	(*Part 17 Present*)
		Part_Present17FB(
			Sensor_Input:= N03.I.0,
			On_Trigger1:= Enable_Motion AND In_Auto AND NOT Unload_Complete AND (Model_ID <> 1) AND Repo_Reqs.0,
			On_Trigger2:= TRUE,
			Off_Trigger1:= Dry_Cycle OR (Cycle_Complete  AND NOT Enable_Motion),
			Off_Trigger2:= TRUE,
			Disable_Faults:= Dry_Cycle OR (Weld_Robots_WorkingOK) OR Turntable_Bypassed,
			Fault_Delay:= T#1.5s,
			Status=> Part_Present17,
			Faulted=>  PPFaults.17);

	(*Part 18 Present*)
		Part_Present18FB(
			Sensor_Input:= N03.I.1,
			On_Trigger1:= Enable_Motion AND In_Auto AND NOT Unload_Complete AND (Model_ID>3),
			On_Trigger2:= TRUE,
			Off_Trigger1:= Dry_Cycle OR (Cycle_Complete  AND NOT Enable_Motion),
			Off_Trigger2:= TRUE,
			Disable_Faults:= Dry_Cycle OR (Weld_Robots_WorkingOK) OR Turntable_Bypassed,
			Fault_Delay:= T#1.5s,
			Status=> Part_Present18,
			Faulted=>  PPFaults.18);

	(*Part 19 Present*)
		Part_Present19FB(
			Sensor_Input:= N03.I.2,
			On_Trigger1:= Enable_Motion AND In_Auto AND NOT Unload_Complete AND NOT Welding_Complete,
			On_Trigger2:= TRUE,
			Off_Trigger1:= Dry_Cycle OR (Cycle_Complete  AND NOT Enable_Motion),
			Off_Trigger2:= TRUE,
			Disable_Faults:= Dry_Cycle OR (Weld_Robots_WorkingOK) OR Turntable_Bypassed,
			Fault_Delay:= T#1.5s,
			Status=> Part_Present19,
			Faulted=>  PPFaults.19);

	(*Part 20 Present*)
		Part_Present20FB(
			Sensor_Input:= N03.I.3,
			On_Trigger1:= Enable_Motion AND In_Auto AND NOT Unload_Complete,
			On_Trigger2:= TRUE,
			Off_Trigger1:= Dry_Cycle OR (Cycle_Complete  AND NOT Enable_Motion),
			Off_Trigger2:= TRUE,
			Disable_Faults:= Dry_Cycle OR (Weld_Robots_WorkingOK) OR Turntable_Bypassed,
			Fault_Delay:= T#1.5s,
			Status=> Part_Present20,
			Faulted=>  PPFaults.20);

	(*Part 21 Present*)
		Part_Present21FB(
			Sensor_Input:= N03.I.4,
			On_Trigger1:= Enable_Motion AND In_Auto AND NOT Unload_Complete AND NOT Welding_Complete,
			On_Trigger2:= TRUE,
			Off_Trigger1:= Dry_Cycle OR (Cycle_Complete  AND NOT Enable_Motion),
			Off_Trigger2:= TRUE,
			Disable_Faults:= Dry_Cycle OR (Weld_Robots_WorkingOK) OR Turntable_Bypassed,
			Fault_Delay:= T#1.5s,
			Status=> Part_Present21,
			Faulted=>  PPFaults.21);

	(*Part 22 Present*)
		Part_Present22FB(
			Sensor_Input:= N03.I.5,
			On_Trigger1:= Enable_Motion AND In_Auto AND NOT Unload_Complete AND (Model_ID=3) AND NOT Welding_Complete,
			On_Trigger2:= TRUE,
			Off_Trigger1:= Dry_Cycle OR (Cycle_Complete  AND NOT Enable_Motion),
			Off_Trigger2:= TRUE,
			Disable_Faults:= Dry_Cycle OR (Weld_Robots_WorkingOK) OR Turntable_Bypassed,
			Fault_Delay:= T#1.5s,
			Status=> Part_Present22,
			Faulted=>  PPFaults.22);

	(*Part 23 Present - should always be off, detects wrong part loaded*)
		Part_Present23FB(
			Sensor_Input:= N03.I.6,
			On_Trigger1:= FALSE,
			On_Trigger2:= TRUE,
			Off_Trigger1:= Enable_Motion AND In_Auto AND NOT Unload_Complete,
			Off_Trigger2:= TRUE,
			Disable_Faults:= Dry_Cycle OR (Weld_Robots_WorkingOK) OR Turntable_Bypassed,
			Fault_Delay:= T#1.5s,
			Status=> Part_Present23,
			Faulted=>  PPFaults.23);

	(*Part 24 Present*)
		Part_Present24FB(
			Sensor_Input:= N03.I.7,
			On_Trigger1:= Enable_Motion AND In_Auto AND NOT Unload_Complete AND (Model_ID = 2),
			On_Trigger2:= TRUE,
			Off_Trigger1:= Dry_Cycle OR (Cycle_Complete  AND NOT Enable_Motion),
			Off_Trigger2:= TRUE,
			Disable_Faults:= Dry_Cycle OR (Weld_Robots_WorkingOK) OR Turntable_Bypassed,
			Fault_Delay:= T#1.5s,
			Status=> Part_Present24,
			Faulted=>  PPFaults.24);

	(*Part 25 Present*)
		Part_Present25FB(
			Sensor_Input:= N04.I.0,
			On_Trigger1:= Enable_Motion AND In_Auto AND NOT Unload_Complete,
			On_Trigger2:= TRUE,
			Off_Trigger1:= Dry_Cycle OR (Cycle_Complete  AND NOT Enable_Motion),
			Off_Trigger2:= TRUE,
			Disable_Faults:= Dry_Cycle OR (Weld_Robots_WorkingOK) OR Turntable_Bypassed,
			Fault_Delay:= T#1.5s,
			Status=> Part_Present25,
			Faulted=>  PPFaults.25);

	(*Part 26 Present*)
		Part_Present26FB(
			Sensor_Input:= N04.I.1,
			On_Trigger1:= Enable_Motion AND In_Auto AND NOT Unload_Complete,
			On_Trigger2:= TRUE,
			Off_Trigger1:= Dry_Cycle OR (Cycle_Complete  AND NOT Enable_Motion),
			Off_Trigger2:= TRUE,
			Disable_Faults:= Dry_Cycle OR (Weld_Robots_WorkingOK) OR Turntable_Bypassed,
			Fault_Delay:= T#1.5s,
			Status=> Part_Present26,
			Faulted=>  PPFaults.26);

	(*Part 27 Present*)
		Part_Present27FB(
			Sensor_Input:= N04.I.2,
			On_Trigger1:= Enable_Motion AND In_Auto AND NOT Unload_Complete AND NOT Welding_Complete,
			On_Trigger2:= TRUE,
			Off_Trigger1:= Dry_Cycle OR (Cycle_Complete  AND NOT Enable_Motion),
			Off_Trigger2:= TRUE,
			Disable_Faults:= Dry_Cycle OR (Weld_Robots_WorkingOK) OR Turntable_Bypassed,
			Status=> Part_Present27,
			Faulted=>  PPFaults.27);
			
	(*Part 28 Present*)
		Part_Present28FB(
			Sensor_Input:= N04.I.3,
			On_Trigger1:= Enable_Motion AND In_Auto AND NOT Unload_Complete,
			On_Trigger2:= TRUE,
			Off_Trigger1:= Dry_Cycle OR (Cycle_Complete  AND NOT Enable_Motion),
			Off_Trigger2:= TRUE,
			Disable_Faults:= Dry_Cycle OR (Weld_Robots_WorkingOK) OR Turntable_Bypassed,
			Fault_Delay:= T#1.5s,
			Status=> Part_Present28,
			Faulted=>  PPFaults.28);

	(*Part 29 Present*)
		Part_Present29FB(
			Sensor_Input:= N04.I.4,
			On_Trigger1:= Enable_Motion AND In_Auto AND NOT Unload_Complete,
			On_Trigger2:= TRUE,
			Off_Trigger1:= Dry_Cycle OR (Cycle_Complete  AND NOT Enable_Motion),
			Off_Trigger2:= TRUE,
			Disable_Faults:= Dry_Cycle OR (Weld_Robots_WorkingOK) OR Turntable_Bypassed,
			Fault_Delay:= T#1.5s,
			Status=> Part_Present29,
			Faulted=>  PPFaults.29);

	(*Part 30 Present*)
		Part_Present30FB(
			Sensor_Input:= N04.I.5,
			On_Trigger1:= Enable_Motion AND In_Auto AND NOT Unload_Complete AND (Model_ID=7),
			On_Trigger2:= TRUE,
			Off_Trigger1:= Dry_Cycle OR (Cycle_Complete  AND NOT Enable_Motion),
			Off_Trigger2:= TRUE,
			Disable_Faults:= Dry_Cycle OR (Weld_Robots_WorkingOK) OR Turntable_Bypassed,
			Fault_Delay:= T#1.5s,
			Status=> Part_Present30,
			Faulted=>  PPFaults.30);

	(*Part 31 Present*)
		Part_Present31FB(
			Sensor_Input:= N04.I.6,
			On_Trigger1:= Enable_Motion AND In_Auto AND NOT Unload_Complete AND (Model_ID=6),
			On_Trigger2:= TRUE,
			Off_Trigger1:= Dry_Cycle OR (Cycle_Complete  AND NOT Enable_Motion),
			Off_Trigger2:= TRUE,
			Disable_Faults:= Dry_Cycle OR (Weld_Robots_WorkingOK) OR Turntable_Bypassed,
			Fault_Delay:= T#1.5s,
			Status=> Part_Present31,
			Faulted=>  PPFaults.31);

	(*Part 32 Present*)
		Part_Present32FB(
			Sensor_Input:= N04.I.7,
			On_Trigger1:= Enable_Motion AND In_Auto AND NOT Unload_Complete AND (Model_ID=5),
			On_Trigger2:= TRUE,
			Off_Trigger1:= Dry_Cycle OR (Cycle_Complete  AND NOT Enable_Motion),
			Off_Trigger2:= TRUE,
			Disable_Faults:= Dry_Cycle OR (Weld_Robots_WorkingOK) OR Turntable_Bypassed,
			Fault_Delay:= T#1.5s,
			Status=> Part_Present32,
			Faulted=>  PPFaults1.1);

	(*Part 33 Present*)
		Part_Present33FB(
			Sensor_Input:= N19.I.2,
			On_Trigger1:= Enable_Motion AND In_Auto AND NOT Unload_Complete AND (Model_ID=4),
			On_Trigger2:= TRUE,
			Off_Trigger1:= Dry_Cycle OR (Cycle_Complete  AND NOT Enable_Motion),
			Off_Trigger2:= TRUE,
			Disable_Faults:= Dry_Cycle OR (Weld_Robots_WorkingOK) OR Turntable_Bypassed,
			Fault_Delay:= T#1.5s,
			Status=> Part_Present33,
			Faulted=>  PPFaults1.2);

	(*Part 34 Present*)
		Part_Present34FB(
			Sensor_Input:= N19.I.3,
			On_Trigger1:= Enable_Motion AND In_Auto AND NOT Unload_Complete AND (Model_ID=7),
			On_Trigger2:= TRUE,
			Off_Trigger1:= Dry_Cycle OR (Cycle_Complete  AND NOT Enable_Motion),
			Off_Trigger2:= TRUE,
			Disable_Faults:= Dry_Cycle OR (Weld_Robots_WorkingOK) OR Turntable_Bypassed,
			Fault_Delay:= T#1.5s,
			Status=> Part_Present34,
			Faulted=>  PPFaults1.3);

	(*Part 35 Present*)
		Part_Present35FB(
			Sensor_Input:= N19.I.4,
			On_Trigger1:= Enable_Motion AND In_Auto AND NOT Unload_Complete AND (Model_ID=6),
			On_Trigger2:= TRUE,
			Off_Trigger1:= Dry_Cycle OR (Cycle_Complete  AND NOT Enable_Motion),
			Off_Trigger2:= TRUE,
			Disable_Faults:= Dry_Cycle OR (Weld_Robots_WorkingOK) OR Turntable_Bypassed,
			Fault_Delay:= T#1.5s,
			Status=> Part_Present35,
			Faulted=>  PPFaults1.4);

	(*Part 36 Present*)
		Part_Present36FB(
			Sensor_Input:=  N19.I.5,
			On_Trigger1:= Enable_Motion AND In_Auto AND NOT Unload_Complete AND (Model_ID=5),
			On_Trigger2:= TRUE,
			Off_Trigger1:= Dry_Cycle OR (Cycle_Complete  AND NOT Enable_Motion),
			Off_Trigger2:= TRUE,
			Disable_Faults:= Dry_Cycle OR (Weld_Robots_WorkingOK) OR Turntable_Bypassed,
			Fault_Delay:= T#1.5s,
			Status=> Part_Present36,
			Faulted=>  PPFaults1.5);

	(*Part 37 Present*)
		Part_Present37FB(
			Sensor_Input:=  N19.I.6,
			On_Trigger1:= Enable_Motion AND In_Auto AND NOT Unload_Complete AND (Model_ID=4),
			On_Trigger2:= TRUE,
			Off_Trigger1:= Dry_Cycle OR (Cycle_Complete  AND NOT Enable_Motion),
			Off_Trigger2:= TRUE,
			Disable_Faults:= Dry_Cycle OR (Weld_Robots_WorkingOK) OR Turntable_Bypassed,
			Fault_Delay:= T#1.5s,
			Status=> Part_Present37,
			Faulted=>  PPFaults1.6);

	(*Part 38 Present*)
		Part_Present38FB(
			Sensor_Input:=  N19.I.7,
			On_Trigger1:= Enable_Motion AND In_Auto AND NOT Unload_Complete AND (Model_ID<>3),
			On_Trigger2:= TRUE,
			Off_Trigger1:= Dry_Cycle OR (Cycle_Complete  AND NOT Enable_Motion),
			Off_Trigger2:= TRUE,
			Disable_Faults:= Dry_Cycle OR (Weld_Robots_WorkingOK) OR Turntable_Bypassed,
			Fault_Delay:= T#1.5s,
			Status=> Part_Present38,
			Faulted=>  PPFaults1.7);

(*end*)
END_ACTION

ACTION Robot_Registration:


(*#################################### Register Robots to Tool ##################################*)
(*+++++++++++THIS AREA IS CUSTOM PER INSTALLATION AND WILL HAVE TO BE MODIFIED PER +++++++++++++*)
(*+++++++++++THIS AREA IS CUSTOM PER INSTALLATION AND WILL HAVE TO BE MODIFIED PER +++++++++++++*)
(*NOTE: See Example code in Fix 15 / 16*)
(*NOTE: See Example code in Fix 15 / 16*)

	(*Data From Load Robot(s)*)
	Load_Robots_Clear1:= ((NOT (MAIN.R4.Task_ID_Ack=DropOff_Fix03) OR MAIN.R4.At_Home OR (MAIN.R4.Task_ID_Ack=Pickup_Fix03)) AND MAIN.R4.Clear_Of_EquipInterf3);
	Load_Robots_Clear2:= TRUE;
	Load_Robots_Clear:=Load_Robots_Clear1 AND Load_Robots_Clear2;
	Load_Robots_WorkingOK1:= ((MAIN.R4.Task_ID_Ack=DropOff_Fix03) AND MAIN.R4.Operating);
	Load_Robots_WorkingOK2:= FALSE;
	IF (MAIN.R4.At_EquipInterf2 AND MAIN.R4.Clear_To_Unclamp AND NOT MAIN.R4.At_Pounce)
		THEN
		Load_Robots_UnclampEarly1:= TRUE;
	END_IF;
	Load_Robots_Complete1:= (MAIN.R4.At_EquipInterf3 AND (MAIN.R4.Task_ID_Ack=DropOff_Fix03) AND MAIN.R4.Task_Completed);
	Load_Robots_Complete2:= FALSE;
	Load_Robots_PartInEOAT1:= (EOAT04.Part2_In_EOAT);
	Load_Robots_PartInEOAT2:= FALSE;
	Load_Robots_PartInEOAT2:= FALSE;


	(*Data From Turntable*)
	TurntableA_Clear:= MAIN.R5.Clear_Of_HumanInterf1 AND NOT (MAIN.R5.Task_ID_Ack = Sweep_Fix03);
	TurntableB_Clear:= MAIN.R5.Clear_Of_HumanInterf2 AND NOT (MAIN.R5.Task_ID_Ack = Sweep_Fix04);
	Turntable_Clear:= TurntableA_Clear AND TurntableB_Clear;
	TurntableA_At_Robot:= (MAIN.R5.T03.I.0 AND MAIN.R5.T03.I.1);
	TurntableB_At_Robot:= (MAIN.R5.T03.I.2 AND MAIN.R5.T03.I.3);
	Turntable_WorkingOK:= ((MAIN.R5.Task_ID_Ack=Sweep_Fix03) AND MAIN.R5.At_HumanInterf1) OR ((MAIN.R5.Task_ID_Ack=Sweep_Fix04) AND MAIN.R1.At_HumanInterf2);
	TurntableA_Complete:= MAIN.R5.At_HumanInterf1 AND (MAIN.R5.Task_ID_Ack=Sweep_Fix03) AND MAIN.R5.Task_Completed;
	TurntableB_Complete:= MAIN.R5.At_HumanInterf2 AND (MAIN.R5.Task_ID_Ack=Sweep_Fix04) AND MAIN.R5.Task_Completed;


	(*Data From Seal Robot(s)*)
	Seal_Robots_Clear:= TRUE;
	Seal_Robots_WorkingOK:= FALSE;
	IF FALSE
		THEN
		Seal_Robots_UnclampEarly:= TRUE;
	END_IF;
	Seal_Robots_Complete:= FALSE;


	(*Data From Stud Robot(s)*)
	Stud_Robots_Clear:= TRUE;
	Stud_Robots_WorkingOK:= FALSE;
	IF FALSE
		THEN
		Stud_Robots_UnclampEarly:= TRUE;
	END_IF;
	Stud_Robots_Complete:= FALSE;


	(*Data From Weld Robot(s)*)
	Weld_Robots_Clear:= ((MAIN.R5.Clear_Of_EquipInterf1 AND NOT (MAIN.R5.Task_ID_Ack=Weld_Fix03) AND MAIN.R5.Clear_Of_EquipInterf8 AND NOT (MAIN.R5.Task_ID_Ack>=350)) OR MAIN.R5.At_Home)
					AND ((MAIN.R6.Clear_Of_EquipInterf2 AND NOT (MAIN.R6.Task_ID_Ack=Weld_Fix04) AND MAIN.R6.Clear_Of_EquipInterf8 AND NOT (MAIN.R6.Task_ID_Ack>=350)) OR MAIN.R6.At_Home);
					
	Weld_Robots_WorkingOK:= ((MAIN.R5.Task_ID_Ack=Weld_Fix03) AND MAIN.R5.Operating
						AND (MAIN.R6.Task_ID_Ack=Weld_Fix03) AND MAIN.R6.Operating);
	IF FALSE
		THEN
		Weld_Robots_UnclampEarly:= TRUE;
	END_IF;
	
	Weld_Robots_Complete:= (MAIN.R5.At_EquipInterf1 AND (MAIN.R5.Task_ID_Ack=Weld_Fix03) AND MAIN.R5.Task_Completed)
						AND (MAIN.R6.At_EquipInterf1 AND (MAIN.R6.Task_ID_Ack=Weld_Fix03) AND MAIN.R6.Task_Completed);

	(*Change Robots for Current Fixture functionality*) (*If no MIG robots Set to True.  Example code is in Fix15/16*) 
	Mig_Robots_Ready:= ((Main.R5.Fronius_Mig_HotKey AND Main.R6.Fronius_Mig_HotKey)
						AND (NOT Main.R5.Fronius_IgnitionError AND NOT Main.R6.Fronius_IgnitionError))
						OR (Dry_Cycle);

	(*Data From Unload Robot(s)*)
	Unload_Robots_Clear1:= NOT (MAIN.R4.Task_ID_Ack=PickUp_Fix03) OR MAIN.R4.At_Home;
	Unload_Robots_Clear2:= TRUE;
	Unload_Robots_Clear:= (Unload_Robots_Clear1 AND Unload_Robots_Clear2);
	Unload_Robots_WorkingOK1:= ((MAIN.R4.Task_ID_Ack=PickUp_Fix03) AND MAIN.R4.Operating);
	Unload_Robots_WorkingOK2:= FALSE;
	
	IF (MAIN.R4.At_EquipInterf3 AND MAIN.R4.Clear_To_Unclamp AND NOT MAIN.R4.At_Pounce)
		THEN
		Unload_Robots_UnclampEarly1:= TRUE;
	END_IF;
	IF FALSE
		THEN
		Unload_Robots_UnclampEarly1:= FALSE;
	END_IF;
	
	Unload_Robots_Complete1:= (MAIN.R4.At_EquipInterf3 AND (MAIN.R4.Task_ID_Ack=PickUp_Fix03) AND MAIN.R4.Task_Completed);
	Unload_Robots_Complete2:= FALSE;
	Unload_Robots_EOATEmpty1:= (EOAT04.EOAT_Part1_Empty);
	Unload_Robots_EOATEmpty2:= FALSE;


	(*Amalgumate All Robots Clear of Tool*)
	All_Robots_Clear:= Load_Robots_Clear AND Seal_Robots_Clear AND Stud_Robots_Clear AND Turntable_Clear AND Weld_Robots_Clear AND Unload_Robots_Clear;

	(*Data To All Robots*)
	(*Task ID*)
	IF TurnTableA_At_Robot THEN
	R4_Data.Task_ID[11]:=Task_ID;
	END_IF
	R5_Data.Task_ID[1]:=Task_ID;
	R5_Data.Task_ID[9]:=Task_ID;
	R6_Data.Task_ID[9]:=Task_ID;
	R5_Data.Task_ID[11]:=Task_ID; (*THIS IS FOR WHEN R04 COMES FOR A PICK TO MOVE THE ROBOTS IN A PICK POSITION TLK*)
	R6_Data.Task_ID[11]:=Task_ID; (*THIS IS FOR WHEN R04 COMES FOR A PICK TO MOVE THE ROBOTS IN A PICK POSITION TLK*)

	(*Fix ID*)
	IF TurnTableA_At_Robot THEN
	R4_Data.Fix_ID[11]:=Fix_ID;
	END_IF
	R5_Data.Fix_ID[1]:=Fix_ID;
	R5_Data.Fix_ID[9]:=Fix_ID;
	R6_Data.Fix_ID[9]:=Fix_ID;
	R5_Data.Fix_ID[11]:=Fix_ID; (*THIS IS FOR WHEN R04 COMES FOR A PICK TO MOVE THE ROBOTS IN A PICK POSITION TLK*)
	R6_Data.Fix_ID[11]:=Fix_ID; (*THIS IS FOR WHEN R04 COMES FOR A PICK TO MOVE THE ROBOTS IN A PICK POSITION TLK*)
	
	
	(*Model ID*)
	IF TurnTableA_At_Robot THEN
	R4_Data.Model_ID[11]:=Model_ID;
	END_IF
	R5_Data.Model_ID[1]:=Model_ID;
	R5_Data.Model_ID[9]:=Model_ID;
	R6_Data.Model_ID[9]:=Model_ID;
	R5_Data.Model_ID[11]:=Model_ID; (*THIS IS FOR WHEN R04 COMES FOR A PICK TO MOVE THE ROBOTS IN A PICK POSITION TLK*)
	R6_Data.Model_ID[11]:=Model_ID; (*THIS IS FOR WHEN R04 COMES FOR A PICK TO MOVE THE ROBOTS IN A PICK POSITION TLK*)

	(*Proceed from Pounce*)
	IF TurnTableA_At_Robot THEN
	R4_Data.Proceed_From_Pounce[11]:= Robots_Clear_ToProceed;
	END_IF
	R5_Data.Proceed_From_Pounce[1]:= Robots_Clear_ToProceed;
	R5_Data.Proceed_From_Pounce[9]:= Robots_Clear_ToProceed;
	R6_Data.Proceed_From_Pounce[9]:= Robots_Clear_ToProceed;
	R5_Data.Proceed_From_Pounce[11]:= Robots_Clear_ToProceed; (*THIS IS FOR WHEN R04 COMES FOR A PICK TO MOVE THE ROBOTS IN A PICK POSITION TLK*)
	R6_Data.Proceed_From_Pounce[11]:= Robots_Clear_ToProceed; (*THIS IS FOR WHEN R04 COMES FOR A PICK TO MOVE THE ROBOTS IN A PICK POSITION TLK*)

	(*Complete Acks*)
	IF TurnTableA_At_Robot THEN
	R4_Data.Complete_Ack[11]:=(Unload_Complete1_Ack AND Unload_Robots_WorkingOK1) OR (Load_Complete1_Ack AND Load_Robots_WorkingOK1);;
	END_IF
	R5_Data.Complete_Ack[1]:=(TurnA_Complete_Ack AND TurnTable_WorkingOK);
	R5_Data.Complete_Ack[9]:=(Weld_Complete_Ack AND Weld_Robots_WorkingOK);
	R6_Data.Complete_Ack[9]:=(Weld_Complete_Ack AND Weld_Robots_WorkingOK);
	R5_Data.Complete_Ack[11]:=(Weld_Complete_Ack AND Weld_Robots_WorkingOK); (*THIS IS FOR WHEN R04 COMES FOR A PICK TO MOVE THE ROBOTS IN A PICK POSITION TLK*)
	R6_Data.Complete_Ack[11]:=(Weld_Complete_Ack AND Weld_Robots_WorkingOK); (*THIS IS FOR WHEN R04 COMES FOR A PICK TO MOVE THE ROBOTS IN A PICK POSITION TLK*)

	(*Repo Acks*)
	IF TurnTableA_At_Robot THEN
	R4_Data.PeripheralReq_Ack[11]:= Repo_Ack;
	END_IF
	R5_Data.PeripheralReq_Ack[9]:= Repo_Ack;
	R6_Data.PeripheralReq_Ack[9]:= Repo_Ack;
	R5_Data.PeripheralReq_Ack[11]:= Repo_Ack; (*THIS IS FOR WHEN R04 COMES FOR A PICK TO MOVE THE ROBOTS IN A PICK POSITION TLK*)
	R6_Data.PeripheralReq_Ack[11]:= Repo_Ack; (*THIS IS FOR WHEN R04 COMES FOR A PICK TO MOVE THE ROBOTS IN A PICK POSITION TLK*)

(*%%%%%%%%%%%%%% Call Robots to Tool and Give Them, Task ID, Fixture ID and Model ID %%%%%%%%%%%%%%%%%*)
	(* Perform Call To Tool*)
	Tool_Call_ForLoadRobots1:= Enable_Motion AND (NOT Cell_In_Services OR NOT Load_Robots_Clear1)
						AND Start_Load_Robots1 AND NOT Start_Load_Robots2 AND NOT Start_Weld_Robots AND NOT Start_Seal_Robots AND NOT Start_Stud_Robots
						AND NOT Start_Unload_Robots1 AND NOT Start_Unload_Robots2 AND NOT Start_TurntableA AND NOT Start_TurntableB;
	Tool_Call_ForLoadRobots2:= Enable_Motion AND (NOT Cell_In_Services OR NOT Load_Robots_Clear2)
						AND NOT Start_Load_Robots1 AND Start_Load_Robots2 AND NOT Start_Weld_Robots AND NOT Start_Seal_Robots AND NOT Start_Stud_Robots
						AND NOT Start_Unload_Robots1 AND NOT Start_Unload_Robots2 AND NOT Start_TurntableA AND NOT Start_TurntableB;
	Tool_Call_ForSealRobots:=Enable_Motion AND (NOT Cell_In_Services OR NOT Seal_Robots_Clear)
						AND NOT Start_Load_Robots1 AND NOT Start_Load_Robots2 AND NOT Start_Weld_Robots AND Start_Seal_Robots AND NOT Start_Stud_Robots
						AND NOT Start_Unload_Robots1 AND NOT Start_Unload_Robots2 AND NOT Start_TurntableA AND NOT Start_TurntableB;
	Tool_Call_ForStudRobots:=Enable_Motion AND (NOT Cell_In_Services OR NOT Stud_Robots_Clear)
						AND NOT Start_Load_Robots1 AND NOT Start_Load_Robots2 AND NOT Start_Weld_Robots AND NOT Start_Seal_Robots AND Start_Stud_Robots
						AND NOT Start_Unload_Robots1 AND NOT Start_Unload_Robots2 AND NOT Start_TurntableA AND NOT Start_TurntableB;
	Tool_Call_ForSweepA:= Enable_Motion AND (NOT Cell_In_Services OR NOT TurntableA_Clear)
						AND NOT Start_Load_Robots1 AND NOT Start_Load_Robots2 AND NOT Start_Weld_Robots AND NOT Start_Seal_Robots AND NOT Start_Stud_Robots
						AND NOT Start_Unload_Robots1 AND NOT Start_Unload_Robots2 AND Start_TurntableA AND NOT Start_TurntableB;
	Tool_Call_ForSweepB:= Enable_Motion AND (NOT Cell_In_Services OR NOT TurntableB_Clear)
						AND NOT Start_Load_Robots1 AND NOT Start_Load_Robots2 AND NOT Start_Weld_Robots AND NOT Start_Seal_Robots AND NOT Start_Stud_Robots
						AND NOT Start_Unload_Robots1 AND NOT Start_Unload_Robots2 AND NOT Start_TurntableA AND Start_TurntableB;
	Tool_Call_ForWeldRobots:= Enable_Motion AND (NOT Cell_In_Services OR NOT Weld_Robots_Clear)
						AND NOT Start_Load_Robots1 AND NOT Start_Load_Robots2 AND Start_Weld_Robots AND NOT Start_Seal_Robots AND NOT Start_Stud_Robots
						AND NOT Start_Unload_Robots1 AND NOT Start_Unload_Robots2 AND NOT Start_TurntableA AND NOT Start_TurntableB;
	Tool_Call_ForUnloadRobots1:= Enable_Motion AND (NOT Cell_In_Services OR NOT Unload_Robots_Clear1)
						AND NOT Start_Load_Robots1 AND NOT Start_Load_Robots2 AND NOT Start_Weld_Robots AND NOT Start_Seal_Robots AND NOT Start_Stud_Robots
						AND Start_Unload_Robots1 AND NOT Start_Unload_Robots2 AND NOT Start_TurntableA AND NOT Start_TurntableB;
	Tool_Call_ForUnloadRobots2:= Enable_Motion AND (NOT Cell_In_Services OR NOT Unload_Robots_Clear2)
						AND NOT Start_Load_Robots1 AND NOT Start_Load_Robots2 AND NOT Start_Weld_Robots AND NOT Start_Seal_Robots AND NOT Start_Stud_Robots
						AND NOT Start_Unload_Robots1 AND Start_Unload_Robots2 AND NOT Start_TurntableA AND NOT Start_TurntableB;



	(*Allow Robots to Proceed Into Tool*)
	(*!!!!!This is the final OK to allow Robots Into the Tool Area, So it Better Be Ready!!!!!!!*)
	IF Enable_Motion
		THEN
			IF Load_Robots_Proceed1 AND Load_Robots_WorkingOK1 AND Load_Robots_Clear2 AND Seal_Robots_Clear AND Stud_Robots_Clear AND Turntable_Clear AND Weld_Robots_Clear AND Unload_Robots_Clear
				THEN Robots_Clear_ToProceed:=TRUE;
			ELSIF Load_Robots_Proceed2 AND Load_Robots_WorkingOK2 AND Load_Robots_Clear1 AND Seal_Robots_Clear AND Stud_Robots_Clear AND Turntable_Clear AND Weld_Robots_Clear AND Unload_Robots_Clear
				THEN Robots_Clear_ToProceed:=TRUE;
			ELSIF Seal_Robots_Proceed AND Seal_Robots_WorkingOK AND Load_Robots_Clear AND Stud_Robots_Clear AND Turntable_Clear AND Weld_Robots_Clear AND Unload_Robots_Clear
				THEN Robots_Clear_ToProceed:=TRUE;
			ELSIF Stud_Robots_Proceed AND Stud_Robots_WorkingOK AND Load_Robots_Clear AND Seal_Robots_Clear AND Turntable_Clear AND Weld_Robots_Clear AND Unload_Robots_Clear
				THEN Robots_Clear_ToProceed:=TRUE;
			ELSIF Weld_Robots_Proceed AND Weld_Robots_WorkingOK AND Load_Robots_Clear AND Seal_Robots_Clear AND Stud_Robots_Clear AND Turntable_Clear AND Unload_Robots_Clear
				THEN Robots_Clear_ToProceed:=TRUE;
			ELSIF Unload_Robots_Proceed1 AND Unload_Robots_WorkingOK1 AND Seal_Robots_Clear AND Stud_Robots_Clear AND Turntable_Clear AND Weld_Robots_Clear AND Unload_Robots_Clear2
				THEN Robots_Clear_ToProceed:=TRUE;
			ELSIF Unload_Robots_Proceed2 AND Unload_Robots_WorkingOK2 AND Load_Robots_Clear AND Seal_Robots_Clear AND Stud_Robots_Clear AND Turntable_Clear AND Weld_Robots_Clear AND Unload_Robots_Clear1
				THEN Robots_Clear_ToProceed:=TRUE;
			ELSE Robots_Clear_ToProceed:= FALSE;
			END_IF;
		ELSE Robots_Clear_ToProceed:= FALSE;
	END_IF;

(*+++++++++++++++++++++++++++++++++++++++++++++++ Task Complete Acks ++++++++++++++++++++++++++*)
	(*1st Load Complete Ack*)
	Load_Complete1_Ack:= Load_Robots_Complete1 AND (Load_Complete1 OR Load_Complete);

	(*2nd Load Complete Ack*)
	Load_Complete2_Ack:= Load_Robots_Complete2 AND Load_Complete2;

	(*Seal Complete Ack*)
	Seal_Complete_Ack:= Seal_Robots_Complete AND Sealing_Complete;

	(*Stud Complete Ack*)
	Stud_Complete_Ack:= Stud_Robots_Complete AND Stud_Complete;

	(*Sweep Complete ACK*)
	TurnA_Complete_Ack := TurntableA_Complete AND TurntableA_At_Robot;
	TurnB_Complete_Ack := TurntableB_Complete AND TurntableB_At_Robot;

	(*Weld Complete Ack*)
	Weld_Complete_Ack:= Weld_Robots_Complete AND Welding_Complete;

	(*Unload Complete Ack*)
	Unload_Complete1_Ack:= Unload_Robots_Complete1 AND Unload_Complete;

	(*Unload Complete Ack*)
	Unload_Complete2_Ack:= Unload_Robots_Complete2 AND Unload_Complete;





(*end*)
END_ACTION

ACTION Status_and_Faults:



(*^^^^^^^^^^^^^^^^^^^^^^^^^^^^^^^^^^^^^^ General Visualization ^^^^^^^^^^^^^^^^^^^^^^^^^^^^^^^^^^^^*)
	(*For Ready to Load Indicators*)
		(*Flash when tool should be loaded but load is not complete*)
		IF In_Auto AND Tool_At_Home AND NOT Welding_Complete AND All_Robots_Clear AND NOT All_Sensors_On.2
			THEN
				Ready_To_Load:= Pulse_500mS;
				(*Go solid when tool has been loaded properly*)
				(*Go solid when tool is ready to be unloaded*)
		ELSIF In_Auto AND All_Robots_Clear  AND ((Tool_At_Home AND NOT Welding_Complete AND All_Sensors_On.2 AND NOT Enable_Motion)
			OR (Tool_At_Unload.0 AND Welding_Complete AND (Sealing_Complete OR Sealer_Bypass) AND (Stud_Complete OR Stud_Bypass) AND TurntableA_At_Robot AND NOT All_Sensors_Off))
			THEN
				Ready_To_Load:= TRUE;
		ELSE
				Ready_To_Load:= FALSE;
		END_IF;
	(*For Red Stack Light Indicators*)
		Red_Lamp_Req:= PPFaults<>0 OR CLFaulted.0 OR CLFaulted.4 OR (NOT Sealer_Bypass AND MAIN.SL01.Disp1_Volume_NotOK AND (MAIN.R1.Task_ID_Ack=Seal_Fix01)) OR Load_Seq01.Faulted;


	(*Status Banners*)
		(*1 - Check Parts On Sub Check*)
		IF In_Auto AND NOT In_Manual AND NOT Cycle_Complete AND Tool_At_Load.0
			AND NOT Start_Load_Robots1 AND NOT Start_Load_Robots2 AND NOT Start_Seal_Robots AND NOT Start_Stud_Robots AND NOT Start_TurntableA
			AND NOT Start_TurntableB AND NOT Start_Weld_Robots AND NOT Start_Unload_Robots1 AND NOT Start_Unload_Robots2
			THEN
				IF NOT Dry_Cycle AND NOT All_Sensors_On.0
					THEN Status:= 1;
				ELSIF Dry_Cycle AND NOT Load_Complete1
					THEN Status:=1;
				END_IF;
		END_IF;
		(*2 - Sub Check OK*)
		IF In_Auto AND NOT In_Manual AND NOT Cycle_Complete AND Tool_At_Load.1
			AND NOT Start_Load_Robots1 AND NOT Start_Load_Robots2 AND NOT Start_Seal_Robots AND NOT Start_Stud_Robots AND NOT Start_TurntableA
			AND NOT Start_TurntableB AND NOT Start_Weld_Robots AND NOT Start_Unload_Robots1 AND NOT Start_Unload_Robots2
			THEN
				IF NOT Dry_Cycle AND NOT All_Sensors_On.1
					THEN Status:= 2;
				ELSIF Dry_Cycle AND NOT Load_Complete2
					THEN Status:=2;
				END_IF;
		END_IF;
		(*3 - Load Main Part*)
		IF In_Auto AND NOT In_Manual AND NOT Cycle_Complete AND Tool_At_Load.2 AND TurntableA_At_Robot
			AND NOT Start_Load_Robots1 AND NOT Start_Load_Robots2 AND NOT Start_Seal_Robots AND NOT Start_Stud_Robots AND NOT Start_TurntableA
			AND NOT Start_TurntableB AND NOT Start_Weld_Robots AND NOT Start_Unload_Robots1 AND NOT Start_Unload_Robots2
			THEN
				IF NOT Dry_Cycle AND NOT All_Sensors_On.2
					THEN Status:= 3;
				ELSIF Dry_Cycle AND NOT Load_Complete
					THEN Status:=3;
				END_IF;
		END_IF;
		(*10 - Load Parts Onto Tool*)
		IF In_Auto AND NOT In_Manual AND NOT Cycle_Complete AND Tool_At_Load.0
			AND NOT Start_Load_Robots1 AND NOT Start_Load_Robots2 AND NOT Start_Seal_Robots AND NOT Start_Stud_Robots AND NOT Start_TurntableA
			AND NOT Start_TurntableB AND NOT Start_Weld_Robots AND NOT Start_Unload_Robots1 AND NOT Start_Unload_Robots2
			THEN
				IF NOT Dry_Cycle AND NOT All_Sensors_On.2
					THEN Status:= 10;
				ELSIF Dry_Cycle AND NOT Load_Complete
					THEN Status:=10;
				END_IF;
		END_IF;
		(*11 - Robot(s) Loading*)
		IF ((Start_Load_Robots1 OR  Load_Robots_WorkingOK1) OR (Start_Load_Robots2 OR  Load_Robots_WorkingOK2)) AND In_Auto AND NOT In_Manual
			AND NOT Start_Seal_Robots AND NOT Start_Stud_Robots AND NOT Start_TurntableA
			AND NOT Start_TurntableB AND NOT Start_Weld_Robots AND NOT Start_Unload_Robots1 AND NOT Start_Unload_Robots2
			THEN Status:= 11;
		END_IF;
		(*12 - Parts Loaded OK*)
		IF In_Auto AND NOT In_Manual AND NOT Cycle_Complete
			AND NOT Start_Load_Robots1 AND NOT Start_Load_Robots2 AND NOT Start_Seal_Robots AND NOT Start_Stud_Robots AND NOT Start_TurntableA
			 AND NOT Start_TurntableB AND NOT Start_Weld_Robots AND NOT Start_Unload_Robots1 AND NOT Start_Unload_Robots2
			THEN
				IF (All_Sensors_On.0 AND Tool_At_Load.0) AND NOT Dry_Cycle
					THEN Status:= 12;
				ELSIF Load_Complete
					THEN Status:= 12;
				END_IF;
		END_IF;
		(*19 - Robot(s) Stud*)
		IF (Start_Stud_Robots OR Stud_Robots_WorkingOK) AND In_Auto AND NOT In_Manual
			AND NOT Start_Load_Robots1 AND NOT Start_Load_Robots2 AND NOT Start_Weld_Robots AND NOT Start_Seal_Robots AND NOT Start_TurntableA
			 AND NOT Start_TurntableB AND NOT Start_Unload_Robots1 AND NOT Start_Unload_Robots2
			THEN Status:= 19;
		END_IF;
		(*20 - Robot(s) Sealing*)
		IF (Start_Seal_Robots OR Seal_Robots_WorkingOK) AND In_Auto AND NOT In_Manual
			AND NOT Start_Load_Robots1 AND NOT Start_Load_Robots2 AND NOT Start_Weld_Robots AND NOT Start_Stud_Robots AND NOT Start_TurntableA
			 AND NOT Start_TurntableB AND NOT Start_Unload_Robots1 AND NOT Start_Unload_Robots2
			THEN Status:= 20;
		END_IF;
		(*21 - Robot(s) Welding*)
		IF (Start_Weld_Robots OR Weld_Robots_WorkingOK) AND In_Auto AND NOT In_Manual
			AND NOT Start_Load_Robots1 AND NOT Start_Load_Robots2 AND NOT Start_Seal_Robots AND NOT Start_Stud_Robots AND NOT Start_TurntableA
			 AND NOT Start_TurntableB AND NOT Start_Unload_Robots1 AND NOT Start_Unload_Robots2
			THEN Status:= 21;
		END_IF;
		(*22 - Welding Complete / Ready for Unload*)
		IF In_Auto AND NOT In_Manual AND NOT Cycle_Complete AND Welding_Complete
			AND NOT Start_Load_Robots1 AND NOT Start_Load_Robots2 AND NOT Start_Seal_Robots AND NOT Start_Stud_Robots AND NOT Start_TurntableA
			AND NOT Start_TurntableB AND NOT Start_Weld_Robots AND NOT Start_Unload_Robots1 AND NOT Start_Unload_Robots2
			THEN Status:= 22;
		END_IF;
		(*26 - Ready for Rotate*)
		IF (Start_TurntableA OR Start_TurntableB) AND In_Auto AND NOT In_Manual
			AND NOT Start_Load_Robots1 AND NOT Start_Load_Robots2 AND NOT Start_Seal_Robots AND NOT Start_Stud_Robots
			AND NOT Start_Weld_Robots AND NOT Start_Unload_Robots1 AND NOT Start_Unload_Robots2
			THEN Status := 26;
		END_IF;
		(*31 - Robot(s) Unloading*)
		IF (Start_Unload_Robots1 OR Unload_Robots_WorkingOK1 OR Start_Unload_Robots2 OR Unload_Robots_WorkingOK2) AND In_Auto AND NOT In_Manual
			AND NOT Start_Load_Robots1 AND NOT Start_Load_Robots2 AND NOT Start_Seal_Robots AND NOT Start_Stud_Robots AND NOT Start_TurntableA
			AND NOT Start_TurntableB AND NOT Start_Weld_Robots
			THEN Status:= 31;
		END_IF;
		(*32 - Unload Complete*)
		IF In_Auto AND NOT In_Manual AND NOT Cycle_Complete AND Unload_Complete
			AND NOT Start_Load_Robots1 AND NOT Start_Load_Robots2 AND NOT Start_Seal_Robots AND NOT Start_Stud_Robots AND NOT Start_TurntableA
			AND NOT Start_TurntableB AND NOT Start_Weld_Robots AND NOT Start_Unload_Robots1 AND NOT Start_Unload_Robots2
			THEN Status:= 32;
		END_IF;
		(*42 - Cycle Complete*)
		IF In_Auto AND NOT In_Manual AND Cycle_Complete AND All_Sensors_Off
			THEN Status:= 42;
		END_IF;
		(*50 - In Manual*)
		IF In_Manual
			THEN Status:= 50;
		END_IF;
		(*51 - Clamp Fault*)
		IF (CLFaults1>0 OR CLFaults2>0 OR CLFaults3>0 OR CLFaults4>0) AND In_Auto AND NOT In_Manual
			THEN Status:= 51;
		END_IF;
		(*52 - Part Present Sensor Fault*)
		IF PPFaults>0 AND In_Auto AND NOT In_Manual
			THEN Status:= 52;
		END_IF;
		(*53 - Nut Checks Failed Call QA*)
		IF QAChecks_Failed AND In_Auto AND NOT In_Manual
			THEN Status:= 53;
		END_IF;
		(*54 - Sealer Failed Call QA*)
		IF NOT Sealer_Bypass AND (MAIN.SL01.Disp1_Volume_NotOK AND (MAIN.R1.Task_ID_Ack=Seal_Fix01)) AND In_Auto AND NOT In_Manual
			THEN Status:= 54;
		END_IF;
		(*55 - Load Sequence Fault Call QA*)
		IF Load_Seq01.Faulted AND In_Auto AND NOT In_Manual
			THEN Status:= 55;
		END_IF;



(*$$$$$$$$$$$$$$$$$$$$$$$$$$$$$$$$$$$$$$$$$$$$$$$$$$$ Faults $$$$$$$$$$$$$$$$$$$$$$$$$$$$$$$$$$$$$$$$$$$$$$$$$$$$$$$*)

	(*Clamp/Cylider Faults Group 1*)
		IF CLFaults1>0
			THEN CLFaulted.1:=TRUE;
		ELSE
			CLFaulted.1:=FALSE;
		END_IF;
	(*Clamp/Cylider Faults Group 2*)
		IF CLFaults2>0
			THEN CLFaulted.2:=TRUE;
		ELSE
			CLFaulted.2:=FALSE;
		END_IF;
	(*Clamp/Cylider Faults Group 3*)
		IF CLFaults3>0
			THEN CLFaulted.3:=TRUE;
		ELSE
			CLFaulted.3:=FALSE;
		END_IF;
	(*Clamp/Cylinder Faults Group 4 - Reserved Flag for QA Check Motion Faults*)
		IF CLFaults4>0
			THEN CLFaulted.4:=TRUE;
		ELSE
			CLFaulted.4:=FALSE;
		END_IF;
	(*Bit 0 is designated as ANY Clamp Group Faulted*)
	IF CLFaulted.1 OR CLFaulted.2 OR CLFaulted.3
		THEN CLFaulted.0:= TRUE;
	ELSE CLFaulted.0 := FALSE;
	END_IF;

	(*Part Present Sensor Faults*)
		IF (PPFaults>0) OR (PPFaults1>0) OR (PPFaults2>0)
			THEN PPFaulted.0:=TRUE;
		ELSE
			PPFaulted.0:=FALSE;
		END_IF;
























(*end*)
END_ACTION

ACTION Task_Fix_Model_IDs:


	(*Develop Task IDs - See Global Variable, "TaskID_Record"*)

	IF (Start_Load_Robots1 OR Start_Load_Robots2) AND Enable_Motion
		THEN Task_ID:= Dropoff_Fix03;
	ELSIF Start_Seal_Robots AND Enable_Motion
		THEN Task_ID:= Seal_Fix03;
	ELSIF Start_Stud_Robots AND Enable_Motion
		THEN Task_ID:= Stud_Fix03;
	ELSIF Start_Weld_Robots AND Enable_Motion AND (NOT Start_Load_Robots1 AND NOT Start_Load_Robots2) // ADDED this during SIM - RJ
		THEN Task_ID:= Weld_Fix03;
	ELSIF Start_TurnTableA AND Enable_Motion
		THEN Task_ID:= Sweep_Fix03;
	ELSIF (Start_Unload_Robots1 OR Start_Unload_Robots2) AND Enable_Motion
		THEN Task_ID:= Pickup_Fix03;
	ELSE Task_ID:= 0;
	END_IF;

	(*Develop Fixture ID*)
	Fix_ID:= N00.ID;					(*In Future Map Beckhoff Dip Switch Data From IP67 Block to Here*)

	(*Develop Model ID*)
	Model_ID:= Discrete_In.ModelData;
END_ACTION

ACTION Tool_States:


(*+++++++++++THIS AREA IS CUSTOM PER INSTALLATION AND WILL HAVE TO BE MODIFIED PER +++++++++++++*)
(*+++++++++++THIS AREA IS CUSTOM PER INSTALLATION AND WILL HAVE TO BE MODIFIED PER +++++++++++++*)

(*
						 MODEL ID MAP
					 -------------------
				Model ID :  Part ID  :   Tooling ID
					1  	 : 	 504     :     42
					2	 :   524     :	   42
					3	 :   543     :	   47
					4	 :   526     :	   46
					5	 :   536     :	   45
					6	 :   550     :	   44
					7	 :   571     :	   43
	
*)
	

	(*Tooling Position at HOME*)
	Tool_At_HOME:= 
				(((Model_ID=1) OR (Model_ID>3 OR (Model_ID=0)))		(*Model 504, 526, 536, 550, 571*)
				AND Clamp1RETD AND Clamp2RETD AND Clamp3RETD AND Clamp4RETD
				AND Clamp5RETD AND Clamp6RETD AND Clamp7RETD AND Clamp8RETD
				AND Clamp9RETD AND Clamp10RETD AND Clamp11RETD AND Clamp12RETD
				AND Clamp13RETD AND Clamp14RETD AND Clamp15RETD AND Clamp16RETD
				AND Clamp17RETD AND Clamp18RETD AND Clamp19RETD AND Clamp20RETD
				AND Clamp21RETD AND Clamp22RETD AND Pin1ADVD AND Pin2ADVD AND Pin3ADVD AND Pin4ADVD 
				AND Pin5RETD AND Pin6RETD AND Pin7ADVD AND Pin8ADVD AND Pin9ADVD AND Pin10ADVD 
				AND Pin11ADVD AND Pin12ADVD AND Pin13ADVD AND Pin14RETD AND Pin15RETD AND Pin16ADVD AND Pin17ADVD 
				AND Pin18ADVD AND Slide1ADVD AND Slide2ADVD AND Slide3RETD AND Slide4RETD AND Slide5RETD AND Slide6RETD
				AND Slide7RETD AND Slide8RETD AND Slide9RETD AND Slide10ADVD AND Slide11RETD AND Slide12RETD
				AND Slide13ADVD AND Slide14ADVD AND Swing1RETD AND Swing2RETD AND Swing3RETD)
			OR
				((Model_ID=2)		(*524*)
				AND Clamp1RETD AND Clamp2RETD AND Clamp3RETD AND Clamp4RETD
				AND Clamp5RETD AND Clamp6RETD AND Clamp7RETD AND Clamp8RETD
				AND Clamp9RETD AND Clamp10RETD AND Clamp11RETD AND Clamp12RETD
				AND Clamp13RETD AND Clamp14RETD AND Clamp15RETD AND Clamp16RETD
				AND Clamp17RETD AND Clamp18RETD AND Clamp19RETD AND Clamp20RETD
				AND Clamp21RETD AND Clamp22RETD AND Pin1ADVD AND Pin2ADVD AND Pin3ADVD AND Pin4ADVD 
				AND Pin5ADVD AND Pin6RETD AND Pin7ADVD AND Pin8ADVD AND Pin9ADVD AND Pin10ADVD 
				AND Pin11ADVD AND Pin12ADVD AND Pin13ADVD AND Pin14RETD AND Pin15ADVD AND Pin16ADVD AND Pin17ADVD 
				AND Pin18ADVD AND Slide1ADVD AND Slide2ADVD AND Slide3RETD AND Slide4RETD AND Slide5RETD AND Slide6RETD
				AND Slide7RETD AND Slide8RETD AND Slide9RETD AND Slide10ADVD AND Slide11RETD AND Slide12RETD
				AND Slide13ADVD AND Slide14ADVD AND Swing1RETD AND Swing2RETD AND Swing3RETD)
			OR
				((Model_ID=3)		(*543*)
				AND Clamp1RETD AND Clamp2RETD AND Clamp3RETD AND Clamp4RETD
				AND Clamp5RETD AND Clamp6RETD AND Clamp7RETD AND Clamp8RETD
				AND Clamp9RETD AND Clamp10RETD AND Clamp11RETD AND Clamp12RETD
				AND Clamp13RETD AND Clamp14RETD AND Clamp15RETD AND Clamp16RETD
				AND Clamp17RETD AND Clamp18RETD AND Clamp19RETD AND Clamp20RETD
				AND Clamp21RETD AND Clamp22RETD AND Pin1ADVD AND Pin2ADVD AND Pin3ADVD AND Pin4ADVD 
				AND Pin5RETD AND Pin6ADVD AND Pin7ADVD AND Pin8ADVD AND Pin9ADVD AND Pin10ADVD 
				AND Pin11ADVD AND Pin12ADVD AND Pin13ADVD AND Pin14ADVD AND Pin15RETD AND Pin16ADVD AND Pin17ADVD 
				AND Pin18ADVD AND Slide1ADVD AND Slide2ADVD AND Slide3RETD AND Slide4RETD AND Slide5RETD AND Slide6RETD
				AND Slide7RETD AND Slide8RETD AND Slide9RETD AND Slide10ADVD AND Slide11RETD AND Slide12RETD
				AND Slide13ADVD AND Slide14ADVD AND Swing1RETD AND Swing2RETD AND Swing3RETD);

	(*Tooling position to load parts*)
	Tool_At_Load.0:=
				(((Model_ID=1) OR (Model_ID>3))		(*Model 504, 526, 536, 550, 571*)
				AND Clamp1RETD AND Clamp2RETD AND Clamp3RETD AND Clamp4RETD
				AND Clamp5RETD AND Clamp6RETD AND Clamp7RETD AND Clamp8RETD
				AND Clamp9RETD AND Clamp10RETD AND Clamp11RETD AND Clamp12RETD
				AND Clamp13RETD AND Clamp14RETD AND Clamp15RETD AND Clamp16RETD
				AND Clamp17RETD AND Clamp18RETD AND Clamp19RETD AND Clamp20RETD
				AND Clamp21RETD AND Clamp22RETD AND Pin1ADVD AND Pin2ADVD AND Pin3ADVD AND Pin4ADVD 
				AND Pin5RETD AND Pin6RETD AND Pin7ADVD AND Pin8ADVD AND Pin9ADVD AND Pin10ADVD 
				AND Pin11ADVD AND Pin12ADVD AND Pin13ADVD AND Pin14RETD AND Pin15RETD AND Pin16ADVD AND Pin17ADVD 
				AND Pin18ADVD AND Slide1ADVD AND Slide2ADVD AND Slide3RETD AND Slide4RETD AND Slide5RETD AND Slide6RETD
				AND Slide7RETD AND Slide8RETD AND Slide9RETD AND Slide10ADVD AND Slide11RETD AND Slide12RETD
				AND Slide13ADVD AND Slide14ADVD AND Swing1RETD AND Swing2RETD AND Swing3RETD)
			OR
				((Model_ID=2)		(*Model 524*)
				AND Clamp1RETD AND Clamp2RETD AND Clamp3RETD AND Clamp4RETD
				AND Clamp5RETD AND Clamp6RETD AND Clamp7RETD AND Clamp8RETD
				AND Clamp9RETD AND Clamp10RETD AND Clamp11RETD AND Clamp12RETD
				AND Clamp13RETD AND Clamp14RETD AND Clamp15RETD AND Clamp16RETD
				AND Clamp17RETD AND Clamp18RETD AND Clamp19RETD AND Clamp20RETD
				AND Clamp21RETD AND Clamp22RETD AND Pin1ADVD AND Pin2ADVD AND Pin3ADVD AND Pin4ADVD 
				AND Pin5ADVD AND Pin6RETD AND Pin7ADVD AND Pin8ADVD AND Pin9ADVD AND Pin10ADVD 
				AND Pin11ADVD AND Pin12ADVD AND Pin13ADVD AND Pin14RETD AND Pin15ADVD AND Pin16ADVD AND Pin17ADVD 
				AND Pin18ADVD AND Slide1ADVD AND Slide2ADVD AND Slide3RETD AND Slide4RETD AND Slide5RETD AND Slide6RETD
				AND Slide7RETD AND Slide8RETD AND Slide9RETD AND Slide10ADVD AND Slide11RETD AND Slide12RETD
				AND Slide13ADVD AND Slide14ADVD AND Swing1RETD AND Swing2RETD AND Swing3RETD)
			OR
				((Model_ID=3)		(*Model 543*)
				AND Clamp1RETD AND Clamp2RETD AND Clamp3RETD AND Clamp4RETD
				AND Clamp5RETD AND Clamp6RETD AND Clamp7RETD AND Clamp8RETD
				AND Clamp9RETD AND Clamp10RETD AND Clamp11RETD AND Clamp12RETD
				AND Clamp13RETD AND Clamp14RETD AND Clamp15RETD AND Clamp16RETD
				AND Clamp17RETD AND Clamp18RETD AND Clamp19RETD AND Clamp20RETD
				AND Clamp21RETD AND Clamp22RETD AND Pin1ADVD AND Pin2ADVD AND Pin3ADVD AND Pin4ADVD 
				AND Pin5RETD AND Pin6ADVD AND Pin7ADVD AND Pin8ADVD AND Pin9ADVD AND Pin10ADVD 
				AND Pin11ADVD AND Pin12ADVD AND Pin13ADVD AND Pin14ADVD AND Pin15RETD AND Pin16ADVD AND Pin17ADVD 
				AND Pin18ADVD AND Slide1ADVD AND Slide2ADVD AND Slide3RETD AND Slide4RETD AND Slide5RETD AND Slide6RETD
				AND Slide7RETD AND Slide8RETD AND Slide9RETD AND Slide10ADVD AND Slide11RETD AND Slide12RETD
				AND Slide13ADVD AND Slide14ADVD AND Swing1RETD AND Swing2RETD AND Swing3RETD);
	
	(*Tooling position on Loading Complete*)	
	Tool_At_Load.1:= 
				(((Model_ID=1) OR (Model_ID>3))		(*Model 504, 526, 536, 550, 571*)
				AND Clamp1ADVD AND Clamp2ADVD AND Clamp3ADVD AND Clamp4ADVD AND Clamp5ADVD AND Clamp5ADVD AND Clamp5ADVD
				AND Clamp6ADVD AND Clamp7ADVD AND Clamp8ADVD AND Clamp9ADVD AND Clamp10ADVD AND Clamp11ADVD AND Clamp12ADVD
				AND Clamp13ADVD AND Clamp14ADVD AND Clamp15ADVD AND Clamp16ADVD AND Clamp17ADVD AND Clamp18ADVD AND Clamp19ADVD
				AND Clamp20ADVD AND Clamp21ADVD AND Clamp22ADVD AND Pin1ADVD AND Pin2ADVD AND Pin3ADVD AND Pin4ADVD AND Pin5RETD
				AND Pin6RETD AND Pin7ADVD AND Pin8ADVD AND Pin9ADVD AND Pin10ADVD AND Pin11ADVD AND Pin12ADVD AND Pin13ADVD
				AND Pin14RETD AND Pin15RETD AND Pin16ADVD AND Pin17ADVD AND Pin18ADVD AND Slide1ADVD AND Slide2ADVD AND Slide3ADVD
				AND Slide4ADVD AND Slide5ADVD AND Slide6ADVD AND Slide7ADVD AND Slide8ADVD AND Slide9ADVD AND Slide10ADVD AND Slide11ADVD
				AND Slide12ADVD AND Slide13ADVD AND Slide14ADVD AND Swing1ADVD AND Swing2ADVD AND Swing3ADVD)
			OR
				((Model_ID=2)		(*Model 524*)
				AND Clamp1ADVD AND Clamp2ADVD AND Clamp3ADVD AND Clamp4ADVD AND Clamp5ADVD AND Clamp5ADVD AND Clamp5ADVD
				AND Clamp6ADVD AND Clamp7ADVD AND Clamp8ADVD AND Clamp9ADVD AND Clamp10ADVD AND Clamp11ADVD AND Clamp12ADVD
				AND Clamp13ADVD AND Clamp14ADVD AND Clamp15ADVD AND Clamp16ADVD AND Clamp17ADVD AND Clamp18ADVD AND Clamp19ADVD
				AND Clamp20ADVD AND Clamp21ADVD AND Clamp22ADVD AND Pin1ADVD AND Pin2ADVD AND Pin3ADVD AND Pin4ADVD AND Pin5ADVD
				AND Pin6RETD AND Pin7ADVD AND Pin8ADVD AND Pin9ADVD AND Pin10ADVD AND Pin11ADVD AND Pin12ADVD AND Pin13ADVD
				AND Pin14RETD AND Pin15ADVD AND Pin16ADVD AND Pin17ADVD AND Pin18ADVD AND Slide1ADVD AND Slide2ADVD AND Slide3ADVD
				AND Slide4ADVD AND Slide5ADVD AND Slide6ADVD AND Slide7ADVD AND Slide8ADVD AND Slide9ADVD AND Slide10ADVD AND Slide11ADVD
				AND Slide12ADVD AND Slide13ADVD AND Slide14ADVD AND Swing1ADVD AND Swing2ADVD AND Swing3ADVD)
			OR
				((Model_ID=3)		(*Model 543*)
				AND Clamp1ADVD AND Clamp2ADVD AND Clamp3ADVD AND Clamp4ADVD AND Clamp5ADVD AND Clamp5ADVD AND Clamp5ADVD
				AND Clamp6ADVD AND Clamp7ADVD AND Clamp8ADVD AND Clamp9ADVD AND Clamp10ADVD AND Clamp11ADVD AND Clamp12ADVD
				AND Clamp13ADVD AND Clamp14ADVD AND Clamp15ADVD AND Clamp16ADVD AND Clamp17ADVD AND Clamp18ADVD AND Clamp19ADVD
				AND Clamp20ADVD AND Clamp21ADVD AND Clamp22ADVD AND Pin1ADVD AND Pin2ADVD AND Pin3ADVD AND Pin4ADVD AND Pin5RETD
				AND Pin6ADVD AND Pin7ADVD AND Pin8ADVD AND Pin9ADVD AND Pin10ADVD AND Pin11ADVD AND Pin12ADVD AND Pin13ADVD
				AND Pin14ADVD AND Pin15RETD AND Pin16ADVD AND Pin17ADVD AND Pin18ADVD AND Slide1ADVD AND Slide2ADVD AND Slide3ADVD
				AND Slide4ADVD AND Slide5ADVD AND Slide6ADVD AND Slide7ADVD AND Slide8ADVD AND Slide9ADVD AND Slide10ADVD AND Slide11ADVD
				AND Slide12ADVD AND Slide13ADVD AND Slide14ADVD AND Swing1ADVD AND Swing2ADVD AND Swing3ADVD);
	(*Tool Position for Calling in Load Robots*)
	Tool_At_Load.2:=  
				(((Model_ID=1) OR (Model_ID>3))		(*Model 504, 526, 536, 550, 571*)
				AND Clamp1ADVD AND Clamp2ADVD AND Clamp3ADVD AND Clamp4ADVD AND Clamp5ADVD
				AND Clamp6RETD AND Clamp7RETD AND Clamp8RETD AND Clamp9ADVD AND Clamp10ADVD AND Clamp11RETD AND Clamp12ADVD
				AND Clamp13ADVD AND Clamp14ADVD AND Clamp15RETD AND Clamp16ADVD AND Clamp17RETD AND Clamp18ADVD AND Clamp19RETD
				AND Clamp20RETD AND Clamp21ADVD AND Clamp22ADVD AND Pin1ADVD AND Pin2ADVD AND Pin3ADVD AND Pin4ADVD AND Pin5RETD
				AND Pin6RETD AND Pin7ADVD AND Pin8ADVD AND Pin9ADVD AND Pin10ADVD AND Pin11ADVD AND Pin12ADVD AND Pin13ADVD
				AND Pin14RETD AND Pin15RETD AND Pin16ADVD AND Pin17ADVD AND Pin18ADVD AND Slide1ADVD AND Slide2ADVD AND Slide3RETD
				AND Slide4RETD AND Slide5RETD AND Slide6RETD AND Slide7RETD AND Slide8RETD AND Slide9RETD AND Slide10ADVD AND Slide11RETD
				AND Slide12RETD AND Slide13ADVD AND Slide14ADVD AND Swing1RETD AND Swing2RETD AND Swing3RETD)
			OR
				((Model_ID=2)		(*Model 524*)
				AND Clamp1ADVD AND Clamp2ADVD AND Clamp3ADVD AND Clamp4ADVD AND Clamp5ADVD
				AND Clamp6ADVD AND Clamp7RETD AND Clamp8RETD AND Clamp9ADVD AND Clamp10ADVD AND Clamp11RETD AND Clamp12ADVD
				AND Clamp13ADVD AND Clamp14ADVD AND Clamp15RETD AND Clamp16ADVD AND Clamp17RETD AND Clamp18ADVD AND Clamp19RETD
				AND Clamp20ADVD AND Clamp21ADVD AND Clamp22ADVD AND Pin1ADVD AND Pin2ADVD AND Pin3ADVD AND Pin4ADVD AND Pin5ADVD
				AND Pin6RETD AND Pin7ADVD AND Pin8ADVD AND Pin9ADVD AND Pin10ADVD AND Pin11ADVD AND Pin12ADVD AND Pin13ADVD
				AND Pin14RETD AND Pin15ADVD AND Pin16ADVD AND Pin17ADVD AND Pin18ADVD AND Slide1ADVD AND Slide2ADVD AND Slide3RETD
				AND Slide4RETD AND Slide5RETD AND Slide6RETD AND Slide7RETD AND Slide8RETD AND Slide9RETD AND Slide10ADVD AND Slide11RETD
				AND Slide12RETD AND Slide13ADVD AND Slide14ADVD AND Swing1RETD AND Swing2RETD AND Swing3RETD)
			OR
				((Model_ID=3)		(*Model 543*)
				AND Clamp1ADVD AND Clamp2ADVD AND Clamp3ADVD AND Clamp4ADVD AND Clamp5ADVD
				AND Clamp6RETD AND Clamp7RETD AND Clamp8ADVD AND Clamp9ADVD AND Clamp10ADVD AND Clamp11RETD AND Clamp12ADVD
				AND Clamp13ADVD AND Clamp14ADVD AND Clamp15RETD AND Clamp16ADVD AND Clamp17RETD AND Clamp18ADVD AND Clamp19ADVD
				AND Clamp20RETD AND Clamp21ADVD AND Clamp22ADVD AND Pin1ADVD AND Pin2ADVD AND Pin3ADVD AND Pin4ADVD AND Pin5RETD
				AND Pin6ADVD AND Pin7ADVD AND Pin8ADVD AND Pin9ADVD AND Pin10ADVD AND Pin11ADVD AND Pin12ADVD AND Pin13ADVD
				AND Pin14ADVD AND Pin15RETD AND Pin16ADVD AND Pin17ADVD AND Pin18ADVD AND Slide1ADVD AND Slide2ADVD AND Slide3RETD
				AND Slide4RETD AND Slide5RETD AND Slide6RETD AND Slide7RETD AND Slide8RETD AND Slide9RETD AND Slide10ADVD AND Slide11RETD
				AND Slide12RETD AND Slide13ADVD AND Slide14ADVD AND Swing1RETD AND Swing2RETD AND Swing3RETD);
	Tool_At_Load.3:= FALSE;
	Tool_At_Load.4:= FALSE;


	Tool_At_Seal.0:= FALSE;
	Tool_At_Seal.1:= FALSE;
	Tool_At_Seal.2:= FALSE;
	Tool_At_Seal.3:= FALSE;
	Tool_At_Seal.4:= FALSE;


	Tool_At_Stud.0:= FALSE;
	Tool_At_Stud.1:= FALSE;
	Tool_At_Stud.2:= FALSE;
	Tool_At_Stud.3:= FALSE;
	Tool_At_Stud.4:= FALSE;

	(*Tooling position for ready to rotate*)
	Tool_At_Rotate.0:= 
				(((Model_ID=1) OR (Model_ID>3))		(*Model 504, 526, 536, 550, 571*)
				AND Clamp1ADVD AND Clamp2ADVD AND Clamp3ADVD AND Clamp4ADVD AND Clamp5ADVD
				AND Clamp6RETD AND Clamp7RETD AND Clamp8RETD AND Clamp9ADVD AND Clamp10ADVD AND Clamp11RETD AND Clamp12ADVD
				AND Clamp13ADVD AND Clamp14ADVD AND Clamp15RETD AND Clamp16ADVD AND Clamp17RETD AND Clamp18ADVD AND Clamp19RETD
				AND Clamp20RETD AND Clamp21ADVD AND Clamp22ADVD AND Pin1ADVD AND Pin2ADVD AND Pin3ADVD AND Pin4ADVD AND Pin5RETD
				AND Pin6RETD AND Pin7ADVD AND Pin8ADVD AND Pin9ADVD AND Pin10ADVD AND Pin11ADVD AND Pin12ADVD AND Pin13ADVD
				AND Pin14RETD AND Pin15RETD AND Pin16ADVD AND Pin17ADVD AND Pin18ADVD AND Slide1ADVD AND Slide2ADVD AND Slide3RETD
				AND Slide4RETD AND Slide5RETD AND Slide6RETD AND Slide7RETD AND Slide8RETD AND Slide9RETD AND Slide10ADVD AND Slide11RETD
				AND Slide12RETD AND Slide13ADVD AND Slide14ADVD AND Swing1RETD AND Swing2RETD AND Swing3RETD)
			OR
				((Model_ID=2)		(*Model 524*)
				AND Clamp1ADVD AND Clamp2ADVD AND Clamp3ADVD AND Clamp4ADVD AND Clamp5ADVD
				AND Clamp6ADVD AND Clamp7RETD AND Clamp8RETD AND Clamp9ADVD AND Clamp10ADVD AND Clamp11RETD AND Clamp12ADVD
				AND Clamp13ADVD AND Clamp14ADVD AND Clamp15RETD AND Clamp16ADVD AND Clamp17RETD AND Clamp18ADVD AND Clamp19RETD
				AND Clamp20ADVD AND Clamp21ADVD AND Clamp22ADVD AND Pin1ADVD AND Pin2ADVD AND Pin3ADVD AND Pin4ADVD AND Pin5ADVD
				AND Pin6RETD AND Pin7ADVD AND Pin8ADVD AND Pin9ADVD AND Pin10ADVD AND Pin11ADVD AND Pin12ADVD AND Pin13ADVD
				AND Pin14RETD AND Pin15ADVD AND Pin16ADVD AND Pin17ADVD AND Pin18ADVD AND Slide1ADVD AND Slide2ADVD AND Slide3RETD
				AND Slide4RETD AND Slide5RETD AND Slide6RETD AND Slide7RETD AND Slide8RETD AND Slide9RETD AND Slide10ADVD AND Slide11RETD
				AND Slide12RETD AND Slide13ADVD AND Slide14ADVD AND Swing1RETD AND Swing2RETD AND Swing3RETD)
			OR
				((Model_ID=3)		(*Model 543*)
				AND Clamp1ADVD AND Clamp2ADVD AND Clamp3ADVD AND Clamp4ADVD AND Clamp5ADVD
				AND Clamp6RETD AND Clamp7RETD AND Clamp8ADVD AND Clamp9ADVD AND Clamp10ADVD AND Clamp11RETD AND Clamp12ADVD
				AND Clamp13ADVD AND Clamp14ADVD AND Clamp15RETD AND Clamp16ADVD AND Clamp17RETD AND Clamp18ADVD AND Clamp19ADVD
				AND Clamp20RETD AND Clamp21ADVD AND Clamp22ADVD AND Pin1ADVD AND Pin2ADVD AND Pin3ADVD AND Pin4ADVD AND Pin5RETD
				AND Pin6ADVD AND Pin7ADVD AND Pin8ADVD AND Pin9ADVD AND Pin10ADVD AND Pin11ADVD AND Pin12ADVD AND Pin13ADVD
				AND Pin14ADVD AND Pin15RETD AND Pin16ADVD AND Pin17ADVD AND Pin18ADVD AND Slide1ADVD AND Slide2ADVD AND Slide3RETD
				AND Slide4RETD AND Slide5RETD AND Slide6RETD AND Slide7RETD AND Slide8RETD AND Slide9RETD AND Slide10ADVD AND Slide11RETD
				AND Slide12RETD AND Slide13ADVD AND Slide14ADVD AND Swing1RETD AND Swing2RETD AND Swing3RETD);
				
	Tool_At_Rotate.1:= FALSE;
	Tool_At_Rotate.2:= FALSE;
	Tool_At_Rotate.3:= FALSE;
	Tool_At_Rotate.4:= FALSE;

	(*Tooling position for welding*)
	Tool_At_Weld.0:= 
				(((Model_ID=1) OR (Model_ID>3))		(*Model 504, 526, 536, 550, 571*)
				AND Clamp1ADVD AND Clamp2ADVD AND Clamp3ADVD AND Clamp4ADVD AND Clamp5ADVD AND Clamp5ADVD AND Clamp5ADVD
				AND Clamp6RETD AND Clamp7ADVD AND Clamp8RETD AND Clamp9ADVD AND Clamp10ADVD AND Clamp11ADVD AND Clamp12ADVD
				AND Clamp13ADVD AND Clamp14ADVD AND Clamp15ADVD AND Clamp16ADVD AND Clamp17ADVD AND Clamp18ADVD AND Clamp19RETD
				AND Clamp20RETD AND Clamp21ADVD AND Clamp22ADVD AND Pin1ADVD AND Pin2ADVD AND Pin3ADVD AND Pin4ADVD AND Pin5RETD
				AND Pin6RETD AND Pin7ADVD AND Pin8ADVD AND Pin9ADVD AND Pin10ADVD AND Pin11ADVD AND Pin12ADVD AND Pin13ADVD
				AND Pin14RETD AND Pin15RETD AND Pin16ADVD AND Pin17ADVD AND Pin18ADVD AND Slide1ADVD AND Slide2ADVD AND Slide3ADVD
				AND Slide4RETD AND Slide5ADVD AND Slide6ADVD AND Slide7ADVD AND Slide8ADVD AND Slide9ADVD AND Slide10ADVD AND Slide11RETD
				AND Slide12ADVD AND Slide13ADVD AND Slide14ADVD AND Swing1RETD AND Swing2ADVD AND Swing3RETD)
			OR
				((Model_ID=2)		(*Model 524*)
				AND Clamp1ADVD AND Clamp2ADVD AND Clamp3ADVD AND Clamp4ADVD AND Clamp5ADVD AND Clamp5ADVD AND Clamp5ADVD
				AND Clamp6ADVD AND Clamp7ADVD AND Clamp8RETD AND Clamp9ADVD AND Clamp10ADVD AND Clamp11ADVD AND Clamp12ADVD
				AND Clamp13ADVD AND Clamp14ADVD AND Clamp15ADVD AND Clamp16ADVD AND Clamp17ADVD AND Clamp18ADVD AND Clamp19RETD
				AND Clamp20ADVD AND Clamp21ADVD AND Clamp22ADVD AND Pin1ADVD AND Pin2ADVD AND Pin3ADVD AND Pin4ADVD AND Pin5ADVD
				AND Pin6RETD AND Pin7ADVD AND Pin8ADVD AND Pin9ADVD AND Pin10ADVD AND Pin11ADVD AND Pin12ADVD AND Pin13ADVD
				AND Pin14RETD AND Pin15ADVD AND Pin16ADVD AND Pin17ADVD AND Pin18ADVD AND Slide1ADVD AND Slide2ADVD AND Slide3ADVD
				AND Slide4ADVD AND Slide5ADVD AND Slide6ADVD AND Slide7ADVD AND Slide8ADVD AND Slide9ADVD AND Slide10ADVD AND Slide11ADVD
				AND Slide12ADVD AND Slide13ADVD AND Slide14ADVD AND Swing1RETD AND Swing2ADVD AND Swing3RETD)
			OR
				((Model_ID=3)		(*Model 543*)
				AND Clamp1ADVD AND Clamp2ADVD AND Clamp3ADVD AND Clamp4ADVD AND Clamp5ADVD AND Clamp5ADVD AND Clamp5ADVD
				AND Clamp6RETD AND Clamp7ADVD AND Clamp8ADVD AND Clamp9ADVD AND Clamp10ADVD AND Clamp11ADVD AND Clamp12ADVD
				AND Clamp13ADVD AND Clamp14ADVD AND Clamp15ADVD AND Clamp16ADVD AND Clamp17ADVD AND Clamp18ADVD AND Clamp19ADVD
				AND Clamp20RETD AND Clamp21ADVD AND Clamp22ADVD AND Pin1ADVD AND Pin2ADVD AND Pin3ADVD AND Pin4ADVD AND Pin5RETD
				AND Pin6ADVD AND Pin7ADVD AND Pin8ADVD AND Pin9ADVD AND Pin10ADVD AND Pin11ADVD AND Pin12ADVD AND Pin13ADVD
				AND Pin14ADVD AND Pin15RETD AND Pin16ADVD AND Pin17ADVD AND Pin18ADVD AND Slide1ADVD AND Slide2ADVD AND Slide3ADVD
				AND Slide4RETD AND Slide5ADVD AND Slide6ADVD AND Slide7ADVD AND Slide8ADVD AND Slide9ADVD AND Slide10ADVD AND Slide11RETD
				AND Slide12ADVD AND Slide13ADVD AND Slide14ADVD AND Swing1ADVD AND Swing2ADVD AND Swing3ADVD);
	Tool_At_Weld.1:= FALSE;
	Tool_At_Weld.2:= FALSE;
	Tool_At_Weld.3:= FALSE;
	Tool_At_Weld.4:= FALSE;

	(*Tooling position for unload*)
	Tool_At_Unload.0:=Clamp1RETD AND Clamp2RETD AND Clamp3RETD AND Clamp4RETD
				AND Clamp5RETD AND Clamp6RETD AND Clamp7ADVD AND Clamp8RETD
				AND Clamp9RETD AND Clamp10RETD AND Clamp11ADVD AND Clamp12RETD
				AND Clamp13RETD AND Clamp14RETD AND Clamp15ADVD AND Clamp16RETD
				AND Clamp17ADVD AND Clamp18RETD AND Clamp19RETD AND Clamp20RETD
				AND Clamp21RETD AND Clamp22RETD AND Pin1RETD AND Pin2RETD AND Pin3RETD AND Pin4RETD AND Pin5RETD
				AND Pin6RETD AND Pin7RETD AND Pin8RETD AND Pin9RETD AND Pin10RETD AND Pin11RETD AND Pin12RETD 
				AND Pin13RETD AND Pin14RETD AND Pin15RETD AND Pin16RETD AND Pin17RETD AND Pin18RETD
				AND Slide1RETD AND Slide2RETD AND Slide3RETD AND Slide4RETD AND Slide5RETD AND Slide6RETD
				AND Slide7RETD AND Slide8RETD AND Slide9RETD AND Slide10RETD AND Slide11RETD AND Slide12RETD
				AND Slide13RETD AND Slide14RETD AND Swing1RETD AND Swing2RETD AND Swing3RETD;
	
	Tool_At_Unload.1:=Clamp1RETD AND Clamp2RETD AND Clamp3RETD AND Clamp4RETD
				AND Clamp5RETD AND Clamp6RETD AND Clamp7RETD AND Clamp8RETD
				AND Clamp9RETD AND Clamp10RETD AND Clamp11RETD AND Clamp12RETD
				AND Clamp13RETD AND Clamp14RETD AND Clamp15RETD AND Clamp16RETD
				AND Clamp17RETD AND Clamp18RETD AND Clamp19RETD AND Clamp20RETD
				AND Clamp21RETD AND Clamp22RETD AND Pin1RETD AND Pin2RETD AND Pin3RETD AND Pin4RETD AND Pin5RETD
				AND Pin6RETD AND Pin7RETD AND Pin8RETD AND Pin9RETD AND Pin10RETD AND Pin11RETD AND Pin12RETD 
				AND Pin13RETD AND Pin14RETD AND Pin15RETD AND Pin16RETD AND Pin17RETD AND Pin18RETD
				AND Slide1RETD AND Slide2RETD AND Slide3RETD AND Slide4RETD AND Slide5RETD AND Slide6RETD
				AND Slide7RETD AND Slide8RETD AND Slide9RETD AND Slide10RETD AND Slide11RETD AND Slide12RETD
				AND Slide13RETD AND Slide14RETD AND Swing1RETD AND Swing2RETD AND Swing3RETD;
	Tool_At_Unload.2:= FALSE;
	Tool_At_Unload.3:= FALSE;
	Tool_At_Unload.4:= FALSE;







































(*end*)
END_ACTION

ACTION Tool_VBSeq_Repos:
(*+++++++++++THIS AREA IS CUSTOM PER INSTALLATION AND WILL HAVE TO BE MODIFIED PER +++++++++++++*)
(*+++++++++++THIS AREA IS CUSTOM PER INSTALLATION AND WILL HAVE TO BE MODIFIED PER +++++++++++++*)


(*!!!!!!!!!!!!!!!!!!!!!!!!!!!!!!!!!!!!!!!!!! Tool Motion Control !!!!!!!!!!!!!!!!!!!!!!!!!!!!!!!*)

(*----------------------------------------- Clamp / Unclamp Steps -------------------------------*)

(*$$$$$$$$$$$$$$$$$$$$$$$$$$$$$$$$$$ Develop Clamp and Unclamp Interlocks $$$$$$$$$$$$$$$$$$$$$$*)
(* Note: This is one method to create valve bank commands for clamp and unclamp sequencing
you are welcome to use the direct method as well*)


	(*---------------------------------------------------------Start Clamp Sequence---------------------------------------------------------*)
	
	(*First Stage Clamping*)		(*V8, V10 ADV, IF Model 2 then V2 ADV, IF Model 3 then V5 ADV*)
	Clamp_Step.0:= Auto_Run AND NOT Welding_Complete OR (Cycle_Complete AND NOT Tool_At_Home AND All_Sensors_Off);
	
	
	(*Second Stage Clamping*)		(*V7, V9, V11 ADV, IF Model 2 then V1 ADV, IF Model 3 V4 ADV*)
	
	(*Model 504, 526, 536, 550, 571*)
	IF (Model_ID=1) OR (Model_ID>3) THEN		
				Clamp_Step.1:=  Clamp_Step.0 AND (Load_Complete1 OR Load_Complete2) AND
								(*V8*)
								(Pin1ADVD AND Pin2ADVD AND Pin3ADVD AND Pin4ADVD AND Pin7ADVD 
								AND Pin9ADVD AND Pin16ADVD AND Pin17ADVD AND Pin18ADVD AND Slide10ADVD)
								(*V10*)
								AND (Pin8ADVD AND Pin10ADVD AND Pin11ADVD AND Pin12ADVD AND Pin13ADVD 
								AND Slide1ADVD AND Slide2ADVD AND Slide13ADVD AND Slide14ADVD);
		(*Model 524*)						
		ELSIF (Model_ID=2) THEN					
				Clamp_Step.1:=  Clamp_Step.0 AND (Load_Complete1 OR Load_Complete2) AND
								(*V2*)
								(Pin5ADVD AND Pin15ADVD)
								(*V8*)
								AND (Pin1ADVD AND Pin2ADVD AND Pin3ADVD AND Pin4ADVD AND Pin7ADVD 
								AND Pin9ADVD AND Pin16ADVD AND Pin17ADVD AND Pin18ADVD AND Slide10ADVD)
								(*V10*)
								AND (Pin8ADVD AND Pin10ADVD AND Pin11ADVD AND Pin12ADVD AND Pin13ADVD 
								AND Slide1ADVD AND Slide2ADVD AND Slide13ADVD AND Slide14ADVD);
		(*Model 543*)			
		ELSIF (Model_ID=3) THEN					
				Clamp_Step.1:=  Clamp_Step.0 AND (Load_Complete1 OR Load_Complete2) AND 
								(*V5*)
								(Pin6ADVD AND Pin14ADVD)
								(*V8*)
								AND (Pin1ADVD AND Pin2ADVD AND Pin3ADVD AND Pin4ADVD AND Pin7ADVD 
								AND Pin9ADVD AND Pin16ADVD AND Pin17ADVD AND Pin18ADVD AND Slide10ADVD)
								(*V10*)
								AND (Pin8ADVD AND Pin10ADVD AND Pin11ADVD AND Pin12ADVD AND Pin13ADVD 
								AND Slide1ADVD AND Slide2ADVD AND Slide13ADVD AND Slide14ADVD);						
	END_IF

	
	(*Third Stage Clamping*)		(*V13 ADV*)
	
	(*Model 504, 526, 536, 550, 571*)
	IF (Model_ID=1) OR (Model_ID>3) THEN
				Clamp_Step.2:= 	Clamp_Step.1 AND (All_Sensors_On.2 OR Clamp_Step.2) AND Repo_Reqs.0 AND
								(*V7*)
								(Clamp3ADVD AND Clamp18ADVD)
								(*V9*)
								AND (Clamp1ADVD AND Clamp2ADVD AND Clamp4ADVD AND Clamp5ADVD AND Clamp10ADVD 
								AND Clamp14ADVD AND Clamp21ADVD AND Clamp22ADVD)
								(*V11*)
								AND (Clamp9ADVD AND Clamp12ADVD AND Clamp13ADVD AND Clamp16ADVD);

		ELSIF (Model_ID=2) THEN
				Clamp_Step.2:= 	Clamp_Step.1 AND (All_Sensors_On.2 OR Clamp_Step.2) AND Repo_Reqs.0 AND
								(*V7*)
								(Clamp3ADVD AND Clamp18ADVD)
								(*V9*)
								AND (Clamp1ADVD AND Clamp2ADVD AND Clamp4ADVD AND Clamp5ADVD AND Clamp10ADVD 
								AND Clamp14ADVD AND Clamp21ADVD AND Clamp22ADVD)
								(*V11*)
								AND (Clamp9ADVD AND Clamp12ADVD AND Clamp13ADVD AND Clamp16ADVD)
								(*V1*)
								AND (Clamp6ADVD AND Clamp20ADVD);
		ELSIF (Model_ID=3) THEN
				Clamp_Step.2:= 	Clamp_Step.1 AND (All_Sensors_On.2 OR Clamp_Step.2) AND Repo_Reqs.0 AND
								(*V7*)
								(Clamp3ADVD AND Clamp18ADVD)
								(*V9*)
								AND (Clamp1ADVD AND Clamp2ADVD AND Clamp4ADVD AND Clamp5ADVD AND Clamp10ADVD 
								AND Clamp14ADVD AND Clamp21ADVD AND Clamp22ADVD)
								(*V11*)
								AND (Clamp9ADVD AND Clamp12ADVD AND Clamp13ADVD AND Clamp16ADVD)
								(*V4*)
								AND (Clamp8ADVD AND Clamp19ADVD);
	END_IF


	(*Forth Stage Clamping*)		(*V12 ADV, IF Model 2 V3 ADV, IF Model 3 V6 ADV*)
	
	Clamp_Step.3:= Clamp_Step.2 AND Repo_Reqs.0 AND
					(*V13*)
					(Clamp7ADVD AND Clamp11ADVD AND Clamp15ADVD AND Clamp17ADVD);




	(*---------------------------------------------------------Start Unclamp Sequence---------------------------------------------------------*)

	(*First Stage Unclamping*)		(*V7, V9, V11 RET, IF Model 2 V1 RET, IF Model 3 V4 RET*)

	Unclamp_Step.0:= (Welding_Complete AND TurnTableA_At_Robot);


	(*Second Stage Unclamping*)		(*V8, V10 RET, IF Model 2 V2 RET, IF Model 3 V5 RET*)
	(*Model 504, 526, 536, 550, 571*)
	IF (Model_ID=1) OR (Model_ID>3) THEN
			Unclamp_Step.1:= Unclamp_Step.0 AND 
								(*V7*)
								(Clamp3RETD AND Clamp18RETD)
								(*V9*)
								AND (Clamp1RETD AND Clamp2RETD AND Clamp4RETD AND Clamp5RETD AND Clamp10RETD AND Clamp14RETD AND Clamp21RETD AND Clamp22RETD)
								(*V11*)
								AND (Clamp9RETD AND Clamp12RETD AND Clamp13RETD AND Clamp16RETD);
		(*Model 524*)							
		ELSIF (Model_ID=2) THEN
				Unclamp_Step.1:= Unclamp_Step.0 AND 
									(*V7*)
									(Clamp3RETD AND Clamp18RETD)
									(*V9*)
									AND (Clamp1RETD AND Clamp2RETD AND Clamp4RETD AND Clamp5RETD AND Clamp10RETD AND Clamp14RETD AND Clamp21RETD AND Clamp22RETD)
									(*V11*)
									AND (Clamp9RETD AND Clamp12RETD AND Clamp13RETD AND Clamp16RETD)
									(*V1*)
									AND (Clamp6RETD AND Clamp20RETD);
		(*Model 543*)
		ELSIF (Model_ID=3) THEN							
				Unclamp_Step.1:= Unclamp_Step.0 AND 
									(*V7*)
									(Clamp3RETD AND Clamp18RETD)
									(*V9*)
									AND (Clamp1RETD AND Clamp2RETD AND Clamp4RETD AND Clamp5RETD AND Clamp10RETD AND Clamp14RETD AND Clamp21RETD AND Clamp22RETD)
									(*V11*)
									AND (Clamp9RETD AND Clamp12RETD AND Clamp13RETD AND Clamp16RETD)
									(*V4*)
									AND (Clamp8RETD AND Clamp19RETD);
	END_IF

	
	(*Third Stage Unclamping*)		(*V12 RET, IF Model 2 V3 RET, IF Model 3 V6 RET*)
	(*Model 504, 526, 536, 550, 571*)
	IF (Model_ID=1) OR (Model_ID>3) THEN
			Unclamp_Step.2:= Unclamp_Step.1 AND 
						(*V8*)
						(Pin1RETD AND Pin2RETD AND Pin3RETD AND Pin4RETD AND Pin7RETD AND Pin9RETD AND Pin16RETD AND Pin17RETD AND Pin18RETD AND Slide10RETD)
						(*V10*)
						AND (Pin8RETD AND Pin10RETD AND Pin11RETD AND Pin12RETD AND Pin13RETD AND Slide1RETD AND Slide2RETD AND Slide13RETD AND Slide14RETD);
		(*Model 524*)
		ELSIF (Model_ID=2) THEN
				Unclamp_Step.2:= Unclamp_Step.1 AND 
							(*V8*)
							(Pin1RETD AND Pin2RETD AND Pin3RETD AND Pin4RETD AND Pin7RETD AND Pin9RETD AND Pin16RETD AND Pin17RETD AND Pin18RETD AND Slide10RETD)
							(*V10*)
							AND (Pin8RETD AND Pin10RETD AND Pin11RETD AND Pin12RETD AND Pin13RETD AND Slide1RETD AND Slide2RETD AND Slide13RETD AND Slide14RETD)
							(*V2*)
							AND (Pin5RETD AND Pin15RETD);
		(*Model 543*)
		ELSIF (Model_ID=3) THEN
				Unclamp_Step.2:= Unclamp_Step.1 AND 
							(*V8*)
							(Pin1RETD AND Pin2RETD AND Pin3RETD AND Pin4RETD AND Pin7RETD AND Pin9RETD AND Pin16RETD AND Pin17RETD AND Pin18RETD AND Slide10RETD)
							(*V10*)
							AND (Pin8RETD AND Pin10RETD AND Pin11RETD AND Pin12RETD AND Pin13RETD AND Slide1RETD AND Slide2RETD AND Slide13RETD AND Slide14RETD)
							(*V5*)
							AND (Pin6RETD AND Pin14RETD);
	
	END_IF

	(*Fourth Stage Unclamping*)		(*V13 RET*)
	(*Model 504, 526, 536, 550, 571*)
	IF (Model_ID=1) OR (Model_ID>3) THEN
				Unclamp_Step.3:= Unclamp_Step.2 AND Repo_Reqs.1 AND
							(*V12*)
							(Slide3RETD AND Slide5RETD AND Slide6RETD AND Slide7RETD AND Slide8RETD AND Slide9RETD AND Slide12RETD AND Swing2RETD);

		ELSIF (Model_ID=2) THEN
				Unclamp_Step.3:= Unclamp_Step.2 AND Repo_Reqs.1 AND 
							(*V12*)
							(Slide3RETD AND Slide5RETD AND Slide6RETD AND Slide7RETD AND Slide8RETD AND Slide9RETD AND Slide12RETD AND Swing2RETD)
							(*V3*)
							AND (Slide4RETD AND Slide11RETD);
							
							
		ELSIF (Model_ID=3) THEN
				Unclamp_Step.3:= Unclamp_Step.2 AND Repo_Reqs.1 AND 
							(*V12*)
							(Slide3RETD AND Slide5RETD AND Slide6RETD AND Slide7RETD AND Slide8RETD AND Slide9RETD AND Slide12RETD AND Swing2RETD)
							(*V6*)
							AND (Swing1RETD AND Swing3RETD);
							
	END_IF							


(*------------------------------------------- Repositions --------------------------------------*)

	(*Reposition Request#1*)
	IF (MAIN.R4.Peripheral_Req.0 AND (MAIN.R4.Task_ID_Ack=DropOff_Fix03))
		THEN
			Repo_Reqs.0:= TRUE;
	END_IF;

	(*Reposition Request#2*)
	IF (MAIN.R4.Peripheral_Req.1 AND (MAIN.R4.Task_ID_Ack=Pickup_Fix03))
		THEN
			Repo_Reqs.1:= TRUE;
	END_IF;

	(*Reposition Request#3*)
	IF FALSE
		THEN
			Repo_Reqs.2:= TRUE;
	END_IF;

	(*Reposition Request#4*)
	IF FALSE
		THEN
			Repo_Reqs.3:= TRUE;
	END_IF;

	(*Reposition Request#5*)
	IF FALSE
		THEN
			Repo_Reqs.4:= TRUE;
	END_IF;

	(*Reposition Request#6*)
	IF FALSE
		THEN
			Repo_Reqs.5:= TRUE;
	END_IF;

	(*Reposition Request#7*)
	IF FALSE
		THEN
			Repo_Reqs.6:= TRUE;
	END_IF;

	(*Reposition Request#8*)
	IF FALSE
		THEN
			Repo_Reqs.7:= TRUE;
	END_IF;

	(*Reset All Reposition Acks At the End Of Cycle*)
	IF Cycle_Complete
		THEN
			Repo_Reqs:= 0;
	END_IF;

(*------------------------- Reposition Acks ---------------------*)
	Repo_Ack.0:= Repo_Reqs.0 AND All_Sensors_On.2 AND Tool_At_Weld.0;
	Repo_Ack.1:= Repo_Reqs.1 AND All_Sensors_On.8 AND Tool_At_Unload.1;
	Repo_Ack.2:= Repo_Reqs.2 AND FALSE;
	Repo_Ack.3:= Repo_Reqs.3 AND FALSE;
	Repo_Ack.4:= Repo_Reqs.4 AND FALSE;
	Repo_Ack.5:= Repo_Reqs.5 AND FALSE;
	Repo_Ack.6:= Repo_Reqs.6 AND FALSE;
	Repo_Ack.7:= Repo_Reqs.7 AND FALSE;
END_ACTION

ACTION ValveBank1:


(*+++++++++++THIS AREA IS CUSTOM PER INSTALLATION AND WILL HAVE TO BE MODIFIED PER +++++++++++++*)
(*+++++++++++THIS AREA IS CUSTOM PER INSTALLATION AND WILL HAVE TO BE MODIFIED PER +++++++++++++*)
(*+++++++++++THIS AREA IS CUSTOM PER INSTALLATION AND WILL HAVE TO BE MODIFIED PER +++++++++++++*)

(*+++++++++++VALVE BANK 1 +++++++++++++*)
(*+++++++++++VALVE BANK 1 +++++++++++++*)
(*+++++++++++VALVE BANK 1 +++++++++++++*)


	(*Valve 1, Model 524 ONLY*)
	(*Clamp #6, 20*)
		Valve1FB
			(
			Enable_Motion:= Enable_Motion,
			Enable_Latch:= TRUE,					(*Enabling Runs Valve as detent type (maintained solenoids*)
			Enable_SideA_PreCharge:= FALSE,		(*Enabling Turns Side A PreCharge Active, reset when Side B is energized in Auto*)
			Enable_SideB_PreCharge:= FALSE,		(*Enabling Turns Side B PreCharge Active, reset when Side A is energized in Auto*)
			PreCharge_Time:= T#0.1S,
			Enable_Auto_Commands:= In_Auto,
			Enable_Manual_Commands:= In_Manual AND (All_Robots_Clear OR TurntableB_At_Robot),  (*TLK ADDED OR*)
			In_Manual_SideA_Command:= Discrete_In.ManReqs.0,
			In_Manual_SideB_Command:= (Discrete_In.ManReqs.1 OR Discrete_In.Go_Home),
			SideA_Indicator:= (Clamp6ADVD AND Clamp20ADVD),
			SideB_Indicator:= (Clamp6RETD AND Clamp20RETD) OR Manual_Ind_HomePrompt,
			TurnOn_SideA_SOL=> N100.Q.0,
			TurnOn_SideB_SOL=> N100.Q.1,
			TurnOn_SideA_Indicator=> Manual_Indicators1.0,
			TurnOn_SideB_Indicator=> Manual_Indicators1.1
			 );
	IF (Model_ID=2) THEN		 
			Valve1FB.In_Auto_SideA_Command:= Clamp_Step.1 AND NOT Unclamp_Step.0;
			Valve1FB.In_Auto_SideB_Command:= Unclamp_Step.0 
										OR ((TurntableA_At_Robot OR Turntable_Bypassed) AND All_Sensors_Off AND Weld_Robots_Clear);
		ELSE
			Valve1FB.In_Auto_SideA_Command:= FALSE;
			Valve1FB.In_Auto_SideB_Command:= TRUE;
		END_IF

	(*Valve 2, Model 524 ONLY*)
	(*Pin #5, 15*)
		Valve2FB
			(
			Enable_Motion:= Enable_Motion,
			Enable_Latch:= TRUE,					(*Enabling Runs Valve as detent type (maintained solenoids*)
			Enable_SideA_PreCharge:= FALSE,		(*Enabling Turns Side A PreCharge Active, reset when Side B is energized in Auto*)
			Enable_SideB_PreCharge:= FALSE,		(*Enabling Turns Side B PreCharge Active, reset when Side A is energized in Auto*)
			PreCharge_Time:= T#0.10S,
			Enable_Auto_Commands:= In_Auto,
			Enable_Manual_Commands:= In_Manual AND (All_Robots_Clear OR TurntableB_At_Robot),  (*TLK ADDED OR*)
			In_Manual_SideA_Command:=  (Discrete_In.ManReqs.2 OR (Discrete_In.Go_Home AND (Model_ID = 2))),
			In_Manual_SideB_Command:= (Discrete_In.ManReqs.3 OR (Discrete_In.Go_Home AND (Model_ID <> 2))),
			SideA_Indicator:=  Pin5ADVD AND Pin15ADVD,
			SideB_Indicator:= (Pin5RETD AND Pin15RETD) OR Manual_Ind_HomePrompt,
			TurnOn_SideA_SOL=> N100.Q.2,
			TurnOn_SideB_SOL=> N100.Q.3,
			TurnOn_SideA_Indicator=> Manual_Indicators1.2,
			TurnOn_SideB_Indicator=> Manual_Indicators1.3
			 );
	IF (Model_ID=2) THEN		 
			Valve2FB.In_Auto_SideA_Command:= Clamp_Step.0 AND NOT Unclamp_Step.1
										OR ((TurntableA_At_Robot OR Turntable_Bypassed) AND All_Sensors_Off AND Weld_Robots_Clear);
			Valve2FB.In_Auto_SideB_Command:= Unclamp_Step.1;
		ELSE
			Valve2FB.In_Auto_SideA_Command:= FALSE;
			Valve2FB.In_Auto_SideB_Command:= TRUE;
		END_IF

	(*Valve 3, Model 524 ONLY*)
	(*Slide #4, 11*)
		Valve3FB
			(
			Enable_Motion:= Enable_Motion,
			Enable_Latch:= TRUE,					(*Enabling Runs Valve as detent type (maintained solenoids*)
			Enable_SideA_PreCharge:= FALSE,		(*Enabling Turns Side A PreCharge Active, reset when Side B is energized in Auto*)
			Enable_SideB_PreCharge:= FALSE,		(*Enabling Turns Side B PreCharge Active, reset when Side A is energized in Auto*)
			PreCharge_Time:= T#0.10S,
			Enable_Auto_Commands:= In_Auto,
			Enable_Manual_Commands:= In_Manual AND (All_Robots_Clear OR TurntableB_At_Robot),  (*TLK ADDED OR*)
			In_Manual_SideA_Command:= Discrete_In.ManReqs.4,
			In_Manual_SideB_Command:= (Discrete_In.ManReqs.5 OR Discrete_In.Go_Home),
			SideA_Indicator:= Slide4ADVD AND Slide11ADVD,
			SideB_Indicator:= (Slide4RETD AND Slide11RETD) OR Manual_Ind_HomePrompt,
			TurnOn_SideA_SOL=> N100.Q.4,
			TurnOn_SideB_SOL=> N100.Q.5,
			TurnOn_SideA_Indicator=> Manual_Indicators1.4,
			TurnOn_SideB_Indicator=> Manual_Indicators1.5
			 );
	IF (Model_ID=2) THEN
			Valve3FB.In_Auto_SideA_Command:= Clamp_Step.3 AND NOT Unclamp_Step.2;
			Valve3FB.In_Auto_SideB_Command:= Unclamp_Step.2
										OR ((TurntableA_At_Robot OR Turntable_Bypassed) AND All_Sensors_Off AND Weld_Robots_Clear);
		ELSE
			Valve3FB.In_Auto_SideA_Command:= FALSE;
			Valve3FB.In_Auto_SideB_Command:= TRUE;
		END_IF

	(*Valve 4, Model 543 ONLY*)
	(*Clamp #8, 19*)
		Valve4FB
			(
			Enable_Motion:= Enable_Motion,
			Enable_Latch:= TRUE,					(*Enabling Runs Valve as detent type (maintained solenoids*)
			Enable_SideA_PreCharge:= FALSE,		(*Enabling Turns Side A PreCharge Active, reset when Side B is energized in Auto*)
			Enable_SideB_PreCharge:= FALSE,		(*Enabling Turns Side B PreCharge Active, reset when Side A is energized in Auto*)
			PreCharge_Time:= T#0.10S,
			Enable_Auto_Commands:= In_Auto,
			Enable_Manual_Commands:= In_Manual AND (All_Robots_Clear OR TurntableB_At_Robot),  (*TLK ADDED OR*)
			In_Manual_SideA_Command:= Discrete_In.ManReqs.6,
			In_Manual_SideB_Command:= (Discrete_In.ManReqs.7 OR Discrete_In.Go_Home),
			SideA_Indicator:= Clamp8ADVD AND Clamp19ADVD,
			SideB_Indicator:= (Clamp8RETD AND Clamp19RETD) OR Manual_Ind_HomePrompt,
			TurnOn_SideA_SOL=> N100.Q.6,
			TurnOn_SideB_SOL=> N100.Q.7,
			TurnOn_SideA_Indicator=> Manual_Indicators1.6,
			TurnOn_SideB_Indicator=> Manual_Indicators1.7
			 );
	IF (Model_ID=3) THEN
			Valve4FB.In_Auto_SideA_Command:= Clamp_Step.1 AND NOT Unclamp_Step.0;
			Valve4FB.In_Auto_SideB_Command:= Unclamp_Step.0
										OR ((TurntableA_At_Robot OR Turntable_Bypassed) AND All_Sensors_Off AND Weld_Robots_Clear);
		ELSE
			Valve4FB.In_Auto_SideA_Command:= FALSE;
			Valve4FB.In_Auto_SideB_Command:= TRUE;
		END_IF

	(*Valve 5, Model 543 ONLY*)
	(*Pin #6, 14*)
		Valve5FB
			(
			Enable_Motion:= Enable_Motion,
			Enable_Latch:= TRUE,					(*Enabling Runs Valve as detent type (maintained solenoids*)
			Enable_SideA_PreCharge:= FALSE,		(*Enabling Turns Side A PreCharge Active, reset when Side B is energized in Auto*)
			Enable_SideB_PreCharge:= FALSE,		(*Enabling Turns Side B PreCharge Active, reset when Side A is energized in Auto*)
			PreCharge_Time:= T#0.10S,
			Enable_Auto_Commands:= In_Auto,
			Enable_Manual_Commands:= In_Manual AND (All_Robots_Clear OR TurntableB_At_Robot),  (*TLK ADDED OR*)
			In_Manual_SideA_Command:= (Discrete_In.ManReqs.8 OR (Discrete_In.Go_Home AND (Model_ID = 3))),
			In_Manual_SideB_Command:= (Discrete_In.ManReqs.9 OR (Discrete_In.Go_Home AND (Model_ID <> 3))),
			SideA_Indicator:=  Pin6ADVD AND Pin14ADVD,
			SideB_Indicator:= (Pin6RETD AND Pin14RETD) OR Manual_Ind_HomePrompt,
			TurnOn_SideA_SOL=> N100.Q.8,
			TurnOn_SideB_SOL=> N100.Q.9,
			TurnOn_SideA_Indicator=> Manual_Indicators1.8,
			TurnOn_SideB_Indicator=> Manual_Indicators1.9
			 );
	IF (Model_ID=3) THEN		 
			Valve5FB.In_Auto_SideA_Command:= Clamp_Step.0 AND NOT Unclamp_Step.1
										OR ((TurntableA_At_Robot OR Turntable_Bypassed) AND All_Sensors_Off AND Weld_Robots_Clear);
			Valve5FB.In_Auto_SideB_Command:= Unclamp_Step.1;
		ELSE
			Valve5FB.In_Auto_SideA_Command:= FALSE;
			Valve5FB.In_Auto_SideB_Command:= TRUE;
		END_IF

	(*Valve 6, Model 543 ONLY*)
	(*Swing #1, 3*)
		Valve6FB
			(
			Enable_Motion:= Enable_Motion,
			Enable_Latch:= TRUE,					(*Enabling Runs Valve as detent type (maintained solenoids*)
			Enable_SideA_PreCharge:= FALSE,		(*Enabling Turns Side A PreCharge Active, reset when Side B is energized in Auto*)
			Enable_SideB_PreCharge:= FALSE,		(*Enabling Turns Side B PreCharge Active, reset when Side A is energized in Auto*)
			PreCharge_Time:= T#0.10S,
			Enable_Auto_Commands:= In_Auto,
			Enable_Manual_Commands:= In_Manual AND (All_Robots_Clear OR TurntableB_At_Robot),  (*TLK ADDED OR*)
			In_Manual_SideA_Command:= Discrete_In.ManReqs.10,
			In_Manual_SideB_Command:= (Discrete_In.ManReqs.11 OR Discrete_In.Go_Home),
			SideA_Indicator:= Swing1ADVD AND Swing3ADVD,
			SideB_Indicator:= (Swing1RETD AND Swing3RETD) OR Manual_Ind_HomePrompt,
			TurnOn_SideA_SOL=> N100.Q.10,
			TurnOn_SideB_SOL=> N100.Q.11,
			TurnOn_SideA_Indicator=> Manual_Indicators1.10,
			TurnOn_SideB_Indicator=> Manual_Indicators1.11
			 );
	IF (Model_ID=3) THEN
			Valve6FB.In_Auto_SideA_Command:= Clamp_Step.3 AND NOT Unclamp_Step.2;
			Valve6FB.In_Auto_SideB_Command:= Unclamp_Step.2
										OR ((TurntableA_At_Robot OR Turntable_Bypassed) AND All_Sensors_Off AND Weld_Robots_Clear);
		ELSE
			Valve6FB.In_Auto_SideA_Command:= FALSE;
			Valve6FB.In_Auto_SideB_Command:= TRUE;
		END_IF

	(*Valve 7, Common*)
	(*Clamp #3, 18 - Manual Clamps*)
		Valve7FB
			(
			Enable_Motion:= Enable_Motion,
			Enable_Latch:= (TurnTable_WorkingOK OR TurnTableA_At_Robot),					(*Enabling Runs Valve as detent type (maintained solenoids*)
			Enable_SideA_PreCharge:= FALSE,		(*Enabling Turns Side A PreCharge Active, reset when Side B is energized in Auto*)
			Enable_SideB_PreCharge:= FALSE,		(*Enabling Turns Side B PreCharge Active, reset when Side A is energized in Auto*)
			PreCharge_Time:= T#0.10S,
			Enable_Auto_Commands:= In_Auto,
			Enable_Manual_Commands:= In_Manual AND (All_Robots_Clear OR TurntableB_At_Robot),  (*TLK ADDED OR*)
			In_Manual_SideA_Command:= Discrete_In.ManReqs.12,
			In_Manual_SideB_Command:= (Discrete_In.ManReqs.13 OR Discrete_In.Go_Home),
			SideA_Indicator:= Clamp3ADVD AND Clamp18ADVD,
			SideB_Indicator:= (Clamp3RETD AND Clamp18RETD) OR Manual_Ind_HomePrompt,
			TurnOn_SideA_SOL=> N100.Q.12,
			TurnOn_SideB_SOL=> N100.Q.13,
			TurnOn_SideA_Indicator=> Manual_Indicators1.12,
			TurnOn_SideB_Indicator=> Manual_Indicators1.13
			 );
		Valve7FB.In_Auto_SideA_Command:= Clamp_Step.1 AND NOT Unclamp_Step.0;
		Valve7FB.In_Auto_SideB_Command:= Unclamp_Step.0
										OR ((TurntableB_At_Robot OR Turntable_Bypassed) AND All_Sensors_Off AND Weld_Robots_Clear);


	(*Valve 8, Common*)
	(*Pin #1-4, 7, 9, 16-18, Slide #10*)
		Valve8FB
			(
			Enable_Motion:= Enable_Motion,
			Enable_Latch:= TRUE,					(*Enabling Runs Valve as detent type (maintained solenoids*)
			Enable_SideA_PreCharge:= FALSE,		(*Enabling Turns Side A PreCharge Active, reset when Side B is energized in Auto*)
			Enable_SideB_PreCharge:= FALSE,		(*Enabling Turns Side B PreCharge Active, reset when Side A is energized in Auto*)
			PreCharge_Time:= T#0.10S,
			Enable_Auto_Commands:= In_Auto,
			Enable_Manual_Commands:= In_Manual AND (All_Robots_Clear OR TurntableB_At_Robot),  (*TLK ADDED OR*)
			In_Manual_SideA_Command:= (Discrete_In.ManReqs.14 OR Discrete_In.Go_Home),
			In_Manual_SideB_Command:= Discrete_In.ManReqs.15,
			SideA_Indicator:= (Pin1ADVD AND Pin2ADVD AND Pin3ADVD AND Pin4ADVD AND Pin7ADVD AND Pin9ADVD AND Pin16ADVD AND Pin17ADVD AND Pin18ADVD AND Slide10ADVD) OR Manual_Ind_HomePrompt,
			SideB_Indicator:= Pin1RETD AND Pin2RETD AND Pin3RETD AND Pin4RETD AND Pin7RETD AND Pin9RETD AND Pin16RETD AND Pin17RETD AND Pin18RETD AND Slide10RETD,
			TurnOn_SideA_SOL=> N100.Q.14,
			TurnOn_SideB_SOL=> N100.Q.15,
			TurnOn_SideA_Indicator=> Manual_Indicators1.14,
			TurnOn_SideB_Indicator=> Manual_Indicators1.15
			 );
		Valve8FB.In_Auto_SideA_Command:= Clamp_Step.0 AND NOT Unclamp_Step.1
										OR ((TurntableA_At_Robot OR Turntable_Bypassed) AND All_Sensors_Off AND Weld_Robots_Clear);
		Valve8FB.In_Auto_SideB_Command:= Unclamp_Step.1;


	(*Valve 9, Common*)
	(*Clamp #1, 2, 4, 5, 10, 14, 21, 22*)
		Valve9FB
			(
			Enable_Motion:= Enable_Motion,
			Enable_Latch:= TRUE,					(*Enabling Runs Valve as detent type (maintained solenoids*)
			Enable_SideA_PreCharge:= FALSE,		(*Enabling Turns Side A PreCharge Active, reset when Side B is energized in Auto*)
			Enable_SideB_PreCharge:= FALSE,		(*Enabling Turns Side B PreCharge Active, reset when Side A is energized in Auto*)
			PreCharge_Time:= T#0.10S,
			Enable_Auto_Commands:= In_Auto,
			Enable_Manual_Commands:= In_Manual AND (All_Robots_Clear OR TurntableB_At_Robot),  (*TLK ADDED OR*)
			In_Manual_SideA_Command:= Discrete_In.ManReqs.16,
			In_Manual_SideB_Command:= (Discrete_In.ManReqs.17 OR Discrete_In.Go_Home),
			SideA_Indicator:= Clamp1ADVD AND Clamp2ADVD AND Clamp4ADVD AND Clamp5ADVD AND Clamp10ADVD AND Clamp14ADVD AND Clamp21ADVD AND Clamp22ADVD,
			SideB_Indicator:= (Clamp1RETD AND Clamp2RETD AND Clamp4RETD AND Clamp5RETD AND Clamp10RETD AND Clamp14RETD AND Clamp21RETD AND Clamp22RETD) OR Manual_Ind_HomePrompt,
			TurnOn_SideA_SOL=> N100.Q.16,
			TurnOn_SideB_SOL=> N100.Q.17,
			TurnOn_SideA_Indicator=> Manual_Indicators1.16,
			TurnOn_SideB_Indicator=> Manual_Indicators1.17
			 );
		Valve9FB.In_Auto_SideA_Command:= Clamp_Step.1 AND NOT Unclamp_Step.0;
		Valve9FB.In_Auto_SideB_Command:= Unclamp_Step.0
										OR ((TurntableA_At_Robot OR Turntable_Bypassed) AND All_Sensors_Off AND Weld_Robots_Clear);


	(*Valve 10, Common*)
	(*Pin #8, 10-13, Slide #1, 2, 13, 14*)
		Valve10FB
			(
			Enable_Motion:= Enable_Motion,
			Enable_Latch:= TRUE,					(*Enabling Runs Valve as detent type (maintained solenoids*)
			Enable_SideA_PreCharge:= FALSE,		(*Enabling Turns Side A PreCharge Active, reset when Side B is energized in Auto*)
			Enable_SideB_PreCharge:= FALSE,		(*Enabling Turns Side B PreCharge Active, reset when Side A is energized in Auto*)
			PreCharge_Time:= T#0.10S,
			Enable_Auto_Commands:= In_Auto,
			Enable_Manual_Commands:= In_Manual AND (All_Robots_Clear OR TurntableB_At_Robot),  (*TLK ADDED OR*)
			In_Manual_SideA_Command:= (Discrete_In.ManReqs.18 OR Discrete_In.Go_Home),
			In_Manual_SideB_Command:= Discrete_In.ManReqs.19,
			SideA_Indicator:= (Pin8ADVD AND Pin10ADVD AND Pin11ADVD AND Pin12ADVD AND Pin13ADVD AND Slide1ADVD AND Slide2ADVD AND Slide13ADVD AND Slide14ADVD) OR Manual_Ind_HomePrompt,
			SideB_Indicator:= Pin8RETD AND Pin10RETD AND Pin11RETD AND Pin12RETD AND Pin13RETD AND Slide1RETD AND Slide2RETD AND Slide13RETD AND Slide14RETD,
			TurnOn_SideA_SOL=> N100.Q.18,
			TurnOn_SideB_SOL=> N100.Q.19,
			TurnOn_SideA_Indicator=> Manual_Indicators1.18,
			TurnOn_SideB_Indicator=> Manual_Indicators1.19
			 );
		Valve10FB.In_Auto_SideA_Command:= Clamp_Step.0 AND NOT Unclamp_Step.1
										OR ((TurntableA_At_Robot OR Turntable_Bypassed) AND All_Sensors_Off AND Weld_Robots_Clear);
		Valve10FB.In_Auto_SideB_Command:= Unclamp_Step.1;


	(*Valve 11, Common*)
	(*Clamp #9, 12, 13, 16*)
		Valve11FB
			(
			Enable_Motion:= Enable_Motion,
			Enable_Latch:= TRUE,					(*Enabling Runs Valve as detent type (maintained solenoids*)
			Enable_SideA_PreCharge:= FALSE,		(*Enabling Turns Side A PreCharge Active, reset when Side B is energized in Auto*)
			Enable_SideB_PreCharge:= FALSE,		(*Enabling Turns Side B PreCharge Active, reset when Side A is energized in Auto*)
			PreCharge_Time:= T#0.10S,
			Enable_Auto_Commands:= In_Auto,
			Enable_Manual_Commands:= In_Manual AND (All_Robots_Clear OR TurntableB_At_Robot),  (*TLK ADDED OR*)
			In_Manual_SideA_Command:= Discrete_In.ManReqs.20,
			In_Manual_SideB_Command:= (Discrete_In.ManReqs.21 OR Discrete_In.Go_Home),
			SideA_Indicator:= Clamp9ADVD AND Clamp12ADVD AND Clamp13ADVD AND Clamp16ADVD,
			SideB_Indicator:= (Clamp9RETD AND Clamp12RETD AND Clamp13RETD AND Clamp16RETD) OR Manual_Ind_HomePrompt,
			TurnOn_SideA_SOL=> N100.Q.20,
			TurnOn_SideB_SOL=> N100.Q.21,
			TurnOn_SideA_Indicator=> Manual_Indicators1.20,
			TurnOn_SideB_Indicator=> Manual_Indicators1.21
			 );
		Valve11FB.In_Auto_SideA_Command:= Clamp_Step.1 AND NOT Unclamp_Step.0;
		Valve11FB.In_Auto_SideB_Command:= Unclamp_Step.0
										OR ((TurntableA_At_Robot OR Turntable_Bypassed) AND All_Sensors_Off AND Weld_Robots_Clear);


	(*Valve 12, Common*)
	(*Slide #3, 5, 7-9, 12, Swing #2*)
		Valve12FB
			(
			Enable_Motion:= Enable_Motion,
			Enable_Latch:= TRUE,					(*Enabling Runs Valve as detent type (maintained solenoids*)
			Enable_SideA_PreCharge:= FALSE,		(*Enabling Turns Side A PreCharge Active, reset when Side B is energized in Auto*)
			Enable_SideB_PreCharge:= FALSE,		(*Enabling Turns Side B PreCharge Active, reset when Side A is energized in Auto*)
			PreCharge_Time:= T#0.10S,
			Enable_Auto_Commands:= In_Auto,
			Enable_Manual_Commands:= In_Manual AND (All_Robots_Clear OR TurntableB_At_Robot),  (*TLK ADDED OR*)
			In_Manual_SideA_Command:= Discrete_In.ManReqs.22,
			In_Manual_SideB_Command:= (Discrete_In.ManReqs.23 OR Discrete_In.Go_Home),
			SideA_Indicator:= Slide3ADVD AND Slide5ADVD AND Slide7ADVD AND Slide8ADVD AND Slide9ADVD AND Slide12ADVD AND Swing2ADVD,
			SideB_Indicator:= (Slide3RETD AND Slide5RETD AND Slide7RETD AND Slide8RETD AND Slide9RETD AND Slide12RETD AND Swing2RETD) OR Manual_Ind_HomePrompt,
			TurnOn_SideA_SOL=> N100.Q.22,
			TurnOn_SideB_SOL=> N100.Q.23,
			TurnOn_SideA_Indicator=> Manual_Indicators1.22,
			TurnOn_SideB_Indicator=> Manual_Indicators1.23
			 );
		Valve12FB.In_Auto_SideA_Command:= Clamp_Step.3 AND NOT Unclamp_Step.2;
		Valve12FB.In_Auto_SideB_Command:= Unclamp_Step.2
										OR ((TurntableA_At_Robot OR Turntable_Bypassed) AND All_Sensors_Off AND Weld_Robots_Clear);


	(*Valve 13, Common*)
	(*Clamp #7, 11, 15, 17*)
		Valve13FB
			(
			Enable_Motion:= Enable_Motion,
			Enable_Latch:= TRUE,					(*Enabling Runs Valve as detent type (maintained solenoids*)
			Enable_SideA_PreCharge:= FALSE,		(*Enabling Turns Side A PreCharge Active, reset when Side B is energized in Auto*)
			Enable_SideB_PreCharge:= FALSE,		(*Enabling Turns Side B PreCharge Active, reset when Side A is energized in Auto*)
			PreCharge_Time:= T#0.10S,
			Enable_Auto_Commands:= In_Auto,
			Enable_Manual_Commands:= In_Manual AND (All_Robots_Clear OR TurntableB_At_Robot),  (*TLK ADDED OR*)
			In_Manual_SideA_Command:= Discrete_In.ManReqs.24,
			In_Manual_SideB_Command:= (Discrete_In.ManReqs.25 OR Discrete_In.Go_Home),
			SideA_Indicator:= Clamp7ADVD AND Clamp11ADVD AND Clamp15ADVD AND Clamp17ADVD,
			SideB_Indicator:= (Clamp7RETD AND Clamp11RETD AND Clamp15RETD AND Clamp17RETD) OR Manual_Ind_HomePrompt,
			TurnOn_SideA_SOL=> N100.Q.24,
			TurnOn_SideB_SOL=> N100.Q.25,
			TurnOn_SideA_Indicator=> Manual_Indicators1.24,
			TurnOn_SideB_Indicator=> Manual_Indicators1.25
			 );
		Valve13FB.In_Auto_SideA_Command:= Clamp_Step.2 AND NOT Unclamp_Step.3;
		Valve13FB.In_Auto_SideB_Command:= Unclamp_Step.3
										OR ((TurntableA_At_Robot OR Turntable_Bypassed) AND All_Sensors_Off AND Weld_Robots_Clear);	
		
		
	(*Valve 14, A+B*)
	(*Locks*)
		Valve14FB
			(
			Enable_Motion:= Enable_Motion ,
			Enable_Latch:= FALSE,					(*Enabling Runs Valve as detent type (maintained solenoids*)
			Enable_SideA_PreCharge:= FALSE,		(*Enabling Turns Side A PreCharge Active, reset when Side B is energized in Auto*)
			Enable_SideB_PreCharge:= FALSE,		(*Enabling Turns Side B PreCharge Active, reset when Side A is energized in Auto*)
			PreCharge_Time:= T#0.10S,
			Enable_Auto_Commands:= In_Auto,
			Enable_Manual_Commands:= In_Manual AND (All_Robots_Clear OR TurntableB_At_Robot),
			In_Manual_SideA_Command:= Discrete_In.ManReqs.26,
			In_Manual_SideB_Command:= Discrete_In.ManReqs.27 
										OR (N100.Q.5 AND NOT (Slide4RETD AND Slide11RETD)) 
										OR (N100.Q.15 AND NOT Slide10RETD) 
										OR (N100.Q.19 AND NOT (Slide1RETD AND Slide2RETD AND Slide13RETD AND Slide14RETD))
										OR (N100.Q.23 AND NOT (Slide3RETD AND Slide5RETD AND Slide7RETD AND Slide8RETD AND Slide9RETD AND Slide12RETD))
										OR (N100.Q.28 AND NOT Slide6RETD)
										OR (N100.Q.4 AND NOT (Slide4ADVD AND Slide11ADVD)) 
										OR (N100.Q.14 AND NOT Slide10ADVD) 
										OR (N100.Q.18 AND NOT (Slide1ADVD AND Slide2ADVD AND Slide13ADVD AND Slide14ADVD))
										OR (N100.Q.22 AND NOT (Slide3ADVD AND Slide5ADVD AND Slide7ADVD AND Slide8ADVD AND Slide9ADVD AND Slide12ADVD))
										OR (N100.Q.28 AND NOT Slide6ADVD),
			SideA_Indicator:= FALSE,
			SideB_Indicator:= FALSE,
			TurnOn_SideA_SOL=> N100.Q.26,
			TurnOn_SideB_SOL=> N100.Q.27,
			TurnOn_SideA_Indicator=> Manual_Indicators1.26,
			TurnOn_SideB_Indicator=> Manual_Indicators1.27
			 );
		Valve14FB.In_Auto_SideA_Command:= NOT Valve14FB.In_Auto_SideB_Command;
		Valve14FB.In_Auto_SideB_Command:= (N100.Q.5 AND NOT (Slide4RETD AND Slide11RETD)) 
										OR (N100.Q.15 AND NOT Slide10RETD) 
										OR (N100.Q.19 AND NOT (Slide1RETD AND Slide2RETD AND Slide13RETD AND Slide14RETD))
										OR (N100.Q.23 AND NOT (Slide3RETD AND Slide5RETD AND Slide7RETD AND Slide8RETD AND Slide9RETD AND Slide12RETD))
										OR (N100.Q.29 AND NOT Slide6RETD)
										OR (N100.Q.4 AND NOT (Slide4ADVD AND Slide11ADVD)) 
										OR (N100.Q.14 AND NOT Slide10ADVD) 
										OR (N100.Q.18 AND NOT (Slide1ADVD AND Slide2ADVD AND Slide13ADVD AND Slide14ADVD))
										OR (N100.Q.22 AND NOT (Slide3ADVD AND Slide5ADVD AND Slide7ADVD AND Slide8ADVD AND Slide9ADVD AND Slide12ADVD))
										OR (N100.Q.28 AND NOT Slide6ADVD);



	(*Valve 15, A+B*)
	(*Slide #6*)
		Valve15FB
			(
			Enable_Motion:= Enable_Motion ,
			Enable_Latch:= TRUE,					(*Enabling Runs Valve as detent type (maintained solenoids*)
			Enable_SideA_PreCharge:= FALSE,		(*Enabling Turns Side A PreCharge Active, reset when Side B is energized in Auto*)
			Enable_SideB_PreCharge:= FALSE,		(*Enabling Turns Side B PreCharge Active, reset when Side A is energized in Auto*)
			PreCharge_Time:= T#0.10S,
			Enable_Auto_Commands:= In_Auto,
			Enable_Manual_Commands:= In_Manual AND (All_Robots_Clear OR TurntableB_At_Robot),  (*TLK ADDED OR*)
			In_Manual_SideA_Command:= Discrete_In.ManReqs.28,
			In_Manual_SideB_Command:= Discrete_In.ManReqs.29,
			SideA_Indicator:= Slide6ADVD,
			SideB_Indicator:= Slide6RETD,
			TurnOn_SideA_SOL=> N100.Q.28,
			TurnOn_SideB_SOL=> N100.Q.29,
			TurnOn_SideA_Indicator=> Manual_Indicators1.28,
			TurnOn_SideB_Indicator=> Manual_Indicators1.29
			 );
		Valve15FB.In_Auto_SideA_Command:= Clamp_Step.3 AND NOT Unclamp_Step.2;
		Valve15FB.In_Auto_SideB_Command:= ((TurntableA_At_Robot OR Turntable_Bypassed) AND All_Sensors_Off AND Weld_Robots_Clear);
		
		
(*--------------------------------------------------------------------------------------------------------------------------------------------*)		
(*                                                           Spare Valves                                                                     *)
(*--------------------------------------------------------------------------------------------------------------------------------------------*)


	(*Valve 16, A+B*)
	(*spare*)
		Valve16FB
			(
			Enable_Motion:= Enable_Motion ,
			Enable_Latch:= TRUE,					(*Enabling Runs Valve as detent type (maintained solenoids*)
			Enable_SideA_PreCharge:= FALSE,		(*Enabling Turns Side A PreCharge Active, reset when Side B is energized in Auto*)
			Enable_SideB_PreCharge:= FALSE,		(*Enabling Turns Side B PreCharge Active, reset when Side A is energized in Auto*)
			PreCharge_Time:= T#0.10S,
			Enable_Auto_Commands:= In_Auto,
			Enable_Manual_Commands:= In_Manual AND (All_Robots_Clear OR TurntableB_At_Robot),  (*TLK ADDED OR*)
			In_Manual_SideA_Command:= Discrete_In.ManReqs.30,
			In_Manual_SideB_Command:= Discrete_In.ManReqs.31,
			SideA_Indicator:= FALSE,
			SideB_Indicator:= FALSE,
			TurnOn_SideA_SOL=> N100.Q.30,
			TurnOn_SideB_SOL=> N100.Q.31,
			TurnOn_SideA_Indicator=> Manual_Indicators1.30,
			TurnOn_SideB_Indicator=> Manual_Indicators1.31
			 );
		Valve16FB.In_Auto_SideA_Command:= FALSE;
		Valve16FB.In_Auto_SideB_Command:= FALSE;


























(*end*)
END_ACTION

ACTION ValveBank2:


(*+++++++++++THIS AREA IS CUSTOM PER INSTALLATION AND WILL HAVE TO BE MODIFIED PER +++++++++++++*)
(*+++++++++++THIS AREA IS CUSTOM PER INSTALLATION AND WILL HAVE TO BE MODIFIED PER +++++++++++++*)
(*+++++++++++THIS AREA IS CUSTOM PER INSTALLATION AND WILL HAVE TO BE MODIFIED PER +++++++++++++*)

(*+++++++++++VALVE BANK 2 +++++++++++++*)
(*+++++++++++VALVE BANK 2 +++++++++++++*)
(*+++++++++++VALVE BANK 2 +++++++++++++*)


	(*Valve 17, A+B*)
	(*spare*)
		Valve17FB
			(
			Enable_Motion:= Enable_Motion ,
			Enable_Latch:= TRUE,					(*Enabling Runs Valve as detent type (maintained solenoids*)
			Enable_SideA_PreCharge:= FALSE,		(*Enabling Turns Side A PreCharge Active, reset when Side B is energized in Auto*)
			Enable_SideB_PreCharge:= FALSE,		(*Enabling Turns Side B PreCharge Active, reset when Side A is energized in Auto*)
			PreCharge_Time:= T#0.1S,
			Enable_Auto_Commands:= In_Auto,
			Enable_Manual_Commands:= In_Manual AND All_Robots_Clear,
			In_Manual_SideA_Command:= Discrete_In.ManReqs2.0,
			In_Manual_SideB_Command:= (Discrete_In.ManReqs2.1 OR Discrete_In.Go_Home),
			SideA_Indicator:= FALSE,
			SideB_Indicator:= FALSE,
			TurnOn_SideA_SOL=> N101.Q.0,
			TurnOn_SideB_SOL=> N101.Q.1,
			TurnOn_SideA_Indicator=> Manual_Indicators2.0,
			TurnOn_SideB_Indicator=> Manual_Indicators2.1
			 );
		Valve17FB.In_Auto_SideA_Command:= FALSE;
		Valve17FB.In_Auto_SideB_Command:= FALSE;


	(*Valve 18, A+B*)
	(*spare*)
		Valve18FB
			(
			Enable_Motion:= Enable_Motion ,
			Enable_Latch:= TRUE,					(*Enabling Runs Valve as detent type (maintained solenoids*)
			Enable_SideA_PreCharge:= FALSE,		(*Enabling Turns Side A PreCharge Active, reset when Side B is energized in Auto*)
			Enable_SideB_PreCharge:= FALSE,		(*Enabling Turns Side B PreCharge Active, reset when Side A is energized in Auto*)
			PreCharge_Time:= T#0.10S,
			Enable_Auto_Commands:= In_Auto,
			Enable_Manual_Commands:= In_Manual AND All_Robots_Clear,
			In_Manual_SideA_Command:= Discrete_In.ManReqs2.2,
			In_Manual_SideB_Command:= Discrete_In.ManReqs2.3,
			SideA_Indicator:= FALSE,
			SideB_Indicator:= FALSE,
			TurnOn_SideA_SOL=> N101.Q.2,
			TurnOn_SideB_SOL=> N101.Q.3,
			TurnOn_SideA_Indicator=> Manual_Indicators2.2,
			TurnOn_SideB_Indicator=> Manual_Indicators2.3
			 );
		Valve18FB.In_Auto_SideA_Command:= FALSE;
		Valve18FB.In_Auto_SideB_Command:= FALSE;

	(*Valve 19, A+B*)
	(*spare*)
		Valve19FB
			(
			Enable_Motion:= Enable_Motion ,
			Enable_Latch:= TRUE,					(*Enabling Runs Valve as detent type (maintained solenoids*)
			Enable_SideA_PreCharge:= FALSE,		(*Enabling Turns Side A PreCharge Active, reset when Side B is energized in Auto*)
			Enable_SideB_PreCharge:= FALSE,		(*Enabling Turns Side B PreCharge Active, reset when Side A is energized in Auto*)
			PreCharge_Time:= T#0.10S,
			Enable_Auto_Commands:= In_Auto,
			Enable_Manual_Commands:= In_Manual AND All_Robots_Clear,
			In_Manual_SideA_Command:= Discrete_In.ManReqs2.4,
			In_Manual_SideB_Command:= Discrete_In.ManReqs2.5,
			SideA_Indicator:= FALSE,
			SideB_Indicator:= FALSE,
			TurnOn_SideA_SOL=> N101.Q.4,
			TurnOn_SideB_SOL=> N101.Q.5,
			TurnOn_SideA_Indicator=> Manual_Indicators2.4,
			TurnOn_SideB_Indicator=> Manual_Indicators2.5
			 );
		Valve19FB.In_Auto_SideA_Command:= FALSE;
		Valve19FB.In_Auto_SideB_Command:= FALSE;


	(*Valve 20, A+B*)
	(*spare*)
		Valve20FB
			(
			Enable_Motion:= Enable_Motion ,
			Enable_Latch:= TRUE,					(*Enabling Runs Valve as detent type (maintained solenoids*)
			Enable_SideA_PreCharge:= FALSE,		(*Enabling Turns Side A PreCharge Active, reset when Side B is energized in Auto*)
			Enable_SideB_PreCharge:= FALSE,		(*Enabling Turns Side B PreCharge Active, reset when Side A is energized in Auto*)
			PreCharge_Time:= T#0.10S,
			Enable_Auto_Commands:= In_Auto,
			Enable_Manual_Commands:= In_Manual AND All_Robots_Clear,
			In_Manual_SideA_Command:= Discrete_In.ManReqs2.6,
			In_Manual_SideB_Command:= Discrete_In.ManReqs2.7,
			SideA_Indicator:= FALSE,
			SideB_Indicator:= FALSE,
			TurnOn_SideA_SOL=> N101.Q.6,
			TurnOn_SideB_SOL=> N101.Q.7,
			TurnOn_SideA_Indicator=> Manual_Indicators2.6,
			TurnOn_SideB_Indicator=> Manual_Indicators2.7
			 );
		Valve20FB.In_Auto_SideA_Command:= FALSE;
		Valve20FB.In_Auto_SideB_Command:= FALSE;


	(*Valve 21, A+B*)
	(*spare*)
		Valve21FB
			(
			Enable_Motion:= Enable_Motion ,
			Enable_Latch:= TRUE,					(*Enabling Runs Valve as detent type (maintained solenoids*)
			Enable_SideA_PreCharge:= FALSE,		(*Enabling Turns Side A PreCharge Active, reset when Side B is energized in Auto*)
			Enable_SideB_PreCharge:= FALSE,		(*Enabling Turns Side B PreCharge Active, reset when Side A is energized in Auto*)
			PreCharge_Time:= T#0.10S,
			Enable_Auto_Commands:= In_Auto,
			Enable_Manual_Commands:= In_Manual AND All_Robots_Clear,
			In_Manual_SideA_Command:= Discrete_In.ManReqs2.8,
			In_Manual_SideB_Command:= Discrete_In.ManReqs2.9,
			SideA_Indicator:= FALSE,
			SideB_Indicator:= FALSE,
			TurnOn_SideA_SOL=> N101.Q.8,
			TurnOn_SideB_SOL=> N101.Q.9,
			TurnOn_SideA_Indicator=> Manual_Indicators2.8,
			TurnOn_SideB_Indicator=> Manual_Indicators2.9
			 );
		Valve21FB.In_Auto_SideA_Command:= FALSE;
		Valve21FB.In_Auto_SideB_Command:= FALSE;


	(*Valve 22, A+B*)
	(*spare*)
		Valve22FB
			(
			Enable_Motion:= Enable_Motion ,
			Enable_Latch:= TRUE,					(*Enabling Runs Valve as detent type (maintained solenoids*)
			Enable_SideA_PreCharge:= FALSE,		(*Enabling Turns Side A PreCharge Active, reset when Side B is energized in Auto*)
			Enable_SideB_PreCharge:= FALSE,		(*Enabling Turns Side B PreCharge Active, reset when Side A is energized in Auto*)
			PreCharge_Time:= T#0.10S,
			Enable_Auto_Commands:= In_Auto,
			Enable_Manual_Commands:= In_Manual AND All_Robots_Clear,
			In_Manual_SideA_Command:= Discrete_In.ManReqs2.10,
			In_Manual_SideB_Command:= Discrete_In.ManReqs2.11,
			SideA_Indicator:= FALSE,
			SideB_Indicator:= FALSE,
			TurnOn_SideA_SOL=> N101.Q.10,
			TurnOn_SideB_SOL=> N101.Q.11,
			TurnOn_SideA_Indicator=> Manual_Indicators2.10,
			TurnOn_SideB_Indicator=> Manual_Indicators2.11
			 );
		Valve22FB.In_Auto_SideA_Command:= FALSE;
		Valve22FB.In_Auto_SideB_Command:= FALSE;


	(*Valve 23, A+B*)
	(*spare*)
		Valve23FB
			(
			Enable_Motion:= Enable_Motion ,
			Enable_Latch:= TRUE,					(*Enabling Runs Valve as detent type (maintained solenoids*)
			Enable_SideA_PreCharge:= FALSE,		(*Enabling Turns Side A PreCharge Active, reset when Side B is energized in Auto*)
			Enable_SideB_PreCharge:= FALSE,		(*Enabling Turns Side B PreCharge Active, reset when Side A is energized in Auto*)
			PreCharge_Time:= T#0.10S,
			Enable_Auto_Commands:= In_Auto,
			Enable_Manual_Commands:= In_Manual AND All_Robots_Clear,
			In_Manual_SideA_Command:= Discrete_In.ManReqs2.12,
			In_Manual_SideB_Command:= Discrete_In.ManReqs2.13,
			SideA_Indicator:= FALSE,
			SideB_Indicator:= FALSE,
			TurnOn_SideA_SOL=> N101.Q.12,
			TurnOn_SideB_SOL=> N101.Q.13,
			TurnOn_SideA_Indicator=> Manual_Indicators2.12,
			TurnOn_SideB_Indicator=> Manual_Indicators2.13
			 );
		Valve23FB.In_Auto_SideA_Command:= FALSE;
		Valve23FB.In_Auto_SideB_Command:= FALSE;


	(*Valve 24, A+B*)
	(*spare*)
		Valve24FB
			(
			Enable_Motion:= Enable_Motion ,
			Enable_Latch:= TRUE,					(*Enabling Runs Valve as detent type (maintained solenoids*)
			Enable_SideA_PreCharge:= FALSE,		(*Enabling Turns Side A PreCharge Active, reset when Side B is energized in Auto*)
			Enable_SideB_PreCharge:= FALSE,		(*Enabling Turns Side B PreCharge Active, reset when Side A is energized in Auto*)
			PreCharge_Time:= T#0.10S,
			Enable_Auto_Commands:= In_Auto,
			Enable_Manual_Commands:= In_Manual AND All_Robots_Clear,
			In_Manual_SideA_Command:= Discrete_In.ManReqs2.14,
			In_Manual_SideB_Command:= Discrete_In.ManReqs2.15,
			SideA_Indicator:= FALSE,
			SideB_Indicator:= FALSE,
			TurnOn_SideA_SOL=> N101.Q.14,
			TurnOn_SideB_SOL=> N101.Q.15,
			TurnOn_SideA_Indicator=> Manual_Indicators2.14,
			TurnOn_SideB_Indicator=> Manual_Indicators2.15
			 );
		Valve24FB.In_Auto_SideA_Command:= FALSE;
		Valve24FB.In_Auto_SideB_Command:= FALSE;


	(*Valve 25, A+B*)
	(*spare*)
		Valve25FB
			(
			Enable_Motion:= Enable_Motion ,
			Enable_Latch:= TRUE,					(*Enabling Runs Valve as detent type (maintained solenoids*)
			Enable_SideA_PreCharge:= FALSE,		(*Enabling Turns Side A PreCharge Active, reset when Side B is energized in Auto*)
			Enable_SideB_PreCharge:= FALSE,		(*Enabling Turns Side B PreCharge Active, reset when Side A is energized in Auto*)
			PreCharge_Time:= T#0.10S,
			Enable_Auto_Commands:= In_Auto,
			Enable_Manual_Commands:= In_Manual AND All_Robots_Clear,
			In_Manual_SideA_Command:= Discrete_In.ManReqs2.16,
			In_Manual_SideB_Command:= Discrete_In.ManReqs2.17,
			SideA_Indicator:= FALSE,
			SideB_Indicator:= FALSE,
			TurnOn_SideA_SOL=> N101.Q.16,
			TurnOn_SideB_SOL=> N101.Q.17,
			TurnOn_SideA_Indicator=> Manual_Indicators2.16,
			TurnOn_SideB_Indicator=> Manual_Indicators2.17
			 );
		Valve25FB.In_Auto_SideA_Command:= FALSE;
		Valve25FB.In_Auto_SideB_Command:= FALSE;


	(*Valve 26, A+B*)
	(*spare*)
		Valve26FB
			(
			Enable_Motion:= Enable_Motion ,
			Enable_Latch:= TRUE,					(*Enabling Runs Valve as detent type (maintained solenoids*)
			Enable_SideA_PreCharge:= FALSE,		(*Enabling Turns Side A PreCharge Active, reset when Side B is energized in Auto*)
			Enable_SideB_PreCharge:= FALSE,		(*Enabling Turns Side B PreCharge Active, reset when Side A is energized in Auto*)
			PreCharge_Time:= T#0.10S,
			Enable_Auto_Commands:= In_Auto,
			Enable_Manual_Commands:= In_Manual AND All_Robots_Clear,
			In_Manual_SideA_Command:= Discrete_In.ManReqs2.18,
			In_Manual_SideB_Command:= Discrete_In.ManReqs2.19,
			SideA_Indicator:= FALSE,
			SideB_Indicator:= FALSE,
			TurnOn_SideA_SOL=> N101.Q.18,
			TurnOn_SideB_SOL=> N101.Q.19,
			TurnOn_SideA_Indicator=> Manual_Indicators2.18,
			TurnOn_SideB_Indicator=> Manual_Indicators2.19
			 );
		Valve26FB.In_Auto_SideA_Command:= FALSE;
		Valve26FB.In_Auto_SideB_Command:= FALSE;


	(*Valve 27, A+B*)
	(*spare*)
		Valve27FB
			(
			Enable_Motion:= Enable_Motion ,
			Enable_Latch:= TRUE,					(*Enabling Runs Valve as detent type (maintained solenoids*)
			Enable_SideA_PreCharge:= FALSE,		(*Enabling Turns Side A PreCharge Active, reset when Side B is energized in Auto*)
			Enable_SideB_PreCharge:= FALSE,		(*Enabling Turns Side B PreCharge Active, reset when Side A is energized in Auto*)
			PreCharge_Time:= T#0.10S,
			Enable_Auto_Commands:= In_Auto,
			Enable_Manual_Commands:= In_Manual AND All_Robots_Clear,
			In_Manual_SideA_Command:= Discrete_In.ManReqs2.20,
			In_Manual_SideB_Command:= Discrete_In.ManReqs2.21,
			SideA_Indicator:= FALSE,
			SideB_Indicator:= FALSE,
			TurnOn_SideA_SOL=> N101.Q.20,
			TurnOn_SideB_SOL=> N101.Q.21,
			TurnOn_SideA_Indicator=> Manual_Indicators2.20,
			TurnOn_SideB_Indicator=> Manual_Indicators2.21
			 );
		Valve27FB.In_Auto_SideA_Command:= FALSE;
		Valve27FB.In_Auto_SideB_Command:= FALSE;


	(*Valve 28, A+B*)
	(*spare*)
		Valve28FB
			(
			Enable_Motion:= Enable_Motion ,
			Enable_Latch:= TRUE,					(*Enabling Runs Valve as detent type (maintained solenoids*)
			Enable_SideA_PreCharge:= FALSE,		(*Enabling Turns Side A PreCharge Active, reset when Side B is energized in Auto*)
			Enable_SideB_PreCharge:= FALSE,		(*Enabling Turns Side B PreCharge Active, reset when Side A is energized in Auto*)
			PreCharge_Time:= T#0.10S,
			Enable_Auto_Commands:= In_Auto,
			Enable_Manual_Commands:= In_Manual AND All_Robots_Clear,
			In_Manual_SideA_Command:= Discrete_In.ManReqs2.22,
			In_Manual_SideB_Command:= Discrete_In.ManReqs2.23,
			SideA_Indicator:= FALSE,
			SideB_Indicator:= FALSE,
			TurnOn_SideA_SOL=> N101.Q.22,
			TurnOn_SideB_SOL=> N101.Q.23,
			TurnOn_SideA_Indicator=> Manual_Indicators2.22,
			TurnOn_SideB_Indicator=> Manual_Indicators2.23
			 );
		Valve28FB.In_Auto_SideA_Command:= FALSE;
		Valve28FB.In_Auto_SideB_Command:= FALSE;


	(*Valve 29, A+B*)
	(*spare*)
		Valve29FB
			(
			Enable_Motion:= Enable_Motion ,
			Enable_Latch:= TRUE,					(*Enabling Runs Valve as detent type (maintained solenoids*)
			Enable_SideA_PreCharge:= FALSE,		(*Enabling Turns Side A PreCharge Active, reset when Side B is energized in Auto*)
			Enable_SideB_PreCharge:= FALSE,		(*Enabling Turns Side B PreCharge Active, reset when Side A is energized in Auto*)
			PreCharge_Time:= T#0.10S,
			Enable_Auto_Commands:= In_Auto,
			Enable_Manual_Commands:= In_Manual AND All_Robots_Clear,
			In_Manual_SideA_Command:= Discrete_In.ManReqs2.24,
			In_Manual_SideB_Command:= Discrete_In.ManReqs2.25,
			SideA_Indicator:= FALSE,
			SideB_Indicator:= FALSE,
			TurnOn_SideA_SOL=> N101.Q.24,
			TurnOn_SideB_SOL=> N101.Q.25,
			TurnOn_SideA_Indicator=> Manual_Indicators2.24,
			TurnOn_SideB_Indicator=> Manual_Indicators2.25
			 );
		Valve29FB.In_Auto_SideA_Command:= FALSE;
		Valve29FB.In_Auto_SideB_Command:= FALSE;


	(*Valve 30, A+B*)
	(*spare*)
		Valve30FB
			(
			Enable_Motion:= Enable_Motion ,
			Enable_Latch:= TRUE,					(*Enabling Runs Valve as detent type (maintained solenoids*)
			Enable_SideA_PreCharge:= FALSE,		(*Enabling Turns Side A PreCharge Active, reset when Side B is energized in Auto*)
			Enable_SideB_PreCharge:= FALSE,		(*Enabling Turns Side B PreCharge Active, reset when Side A is energized in Auto*)
			PreCharge_Time:= T#0.10S,
			Enable_Auto_Commands:= In_Auto,
			Enable_Manual_Commands:= In_Manual AND All_Robots_Clear,
			In_Manual_SideA_Command:= Discrete_In.ManReqs2.26,
			In_Manual_SideB_Command:= Discrete_In.ManReqs2.27,
			SideA_Indicator:= FALSE,
			SideB_Indicator:= FALSE,
			TurnOn_SideA_SOL=> N101.Q.26,
			TurnOn_SideB_SOL=> N101.Q.27,
			TurnOn_SideA_Indicator=> Manual_Indicators2.26,
			TurnOn_SideB_Indicator=> Manual_Indicators2.27
			 );
		Valve30FB.In_Auto_SideA_Command:= FALSE;
		Valve30FB.In_Auto_SideB_Command:= FALSE;


